(* CoDeSys 2.3.10.0 project: 20110511_Pantografo_2Ori_VNT15.pr6 *)
(* Libraries: STANDARD.LB6 5.6.98 11:03:02 *)

(* Global variable list: Global_Variables *)
VAR_GLOBAL CONSTANT
	MaxViti: BYTE:= 15;
	MaxFlange: BYTE:= 8;

	PiGreco: 			REAL := 3.14159265358979;					(*180 gradi*)
	PiGreco2: 		REAL:= 6.28318530717958;					(*360 gradi*)
	PiGrecoMezzi: 	REAL:= 1.5707963267949;					(*90 gradi*)
	PiGreco3Mezzi: 	REAL:= 4.71238898038469;					(*270 gradi*)
	Pigreco4i: 		REAL := 0.78539816339744830961566084581988;				(*45 gradi*)
	Pigreco3_8:		REAL:= 1.1780972450961724644234912687298;	(*60 gradi*)
	Rad2Gr:			REAL:= 57.295779513082320876798154814105; (*coeff. di conversione: 360 / (2*Pigreco)*)

	NonSvitabile:	BYTE:=	4;
	Riavvitare:	BYTE:=	3;
	Svitare:		BYTE:=	2;
	Good:		BYTE:=	1;
	NonEffettuata:	BYTE :=	0;

END_VAR
VAR_GLOBAL
	(*Comunicazione PFB*)
	Global_PFBComOK:	BOOL;
	Global_PFBComKO:	BOOL;

	(*Istanze Globali chiamate nel main*)
	Ist_MapA: 	MapA;
	Ist_MapE:	MapE;
	Ist_MapPFB:	MapPFB;


	(*Cicli*)
	Ist_CyclesMatching: 		CyclesMatching;
	Ist_CyclesDataReceiving:	CyclesDataReceiving;


	(*Macthing*)
	Screw: ARRAY [1..MaxViti] OF BOOL; (*array di esiti di metxhing dove l'indice è l'id_vite*)
	Prodotto:		Ricetta; (*ricetta punti vite*)
END_VAR

(* Data type in PAOLO *)
TYPE Avvitatura :
STRUCT
(*	NumMessaggio       : 	BYTE;
       	LunghezzaPacchetto : 	BYTE;
       	CodiceParametro    : 	BYTE;
       	free: 				BYTE;
	Shake:				Handshake;	(*WORD*)
*)
	ID_vite: 			BYTE;			(*identificativo della vite --> valutare il tipo: INT/STRING *)
 	Viti_Totali_Flangia : 	BYTE;
	ID_Flangia:		BYTE;			(*riferimento della flangia di appartenenza*)
	Chiave:			BYTE;			(*riferimento della chiave che va utilizzata su questa vite*)
	ProgAvvitatura: 	BYTE;			(*numero di programma da passare all'avvitatore per avvitate*)
	ProgRiavvitatura: 	BYTE;			(*numero di programma da passare all'avvitatore per riavvitare  *)
	ProgSvitatura:	BYTE;			(*numero di programma da passare all'avvitatore per svitare... se ZERO disabilita svitatura*)
	EsitoAvvitatura:	BYTE;			(*esito avvitatura 0 non effettuata 1 ok 2 scarto 3 svitato*)
(*esitoavvitatura sostituirebbe free2 della struttura scl*)
	Posizione:		Coordinate;
	TolleranzaR: 		REAL;			(*Raggio di tolleranza del punto*)
	TolleranzaZ: 		REAL;			(*Tolleranza Larga  in Altezza per entrare nello stato di Attesa Esito Avvitatura*)
	AltezzaMin:		REAL;			(*Tolleranza stretta Min Max*)
	AltezzaMax:		REAL;
(*       	riserva : ARRAY[76..123] OF BYTE;
*)
END_STRUCT
END_TYPE

(* Data type in PAOLO/ScambioDati/HEADER *)
TYPE Comandi :
STRUCT
	Matching:			BOOL;	(*comando di pantografo enable*)
	TxScrewingData:		BOOL;	(*comando di invio dati avvitatura*)
	RqstScrewingData:	BOOL;	(*comando di richiesta dati avvitatura*)
	ResettaEsitiAvvitature:	BOOL;
END_STRUCT
END_TYPE

(* Data type in PAOLO/ScambioDati/HEADER *)
TYPE CommunicationA :
STRUCT
	BeckMsgNum: 	BYTE;
	EchoPLCLifeBit:	BOOL;
	BeckLifeBit:		BOOL;
	Beck_ACK:		BOOL;
END_STRUCT
END_TYPE

(* Data type in PAOLO/ScambioDati/HEADER *)
TYPE CommunicationE :
STRUCT
	PlcMsgNum:	BYTE;
	PlcLifeBit:	BOOL;
	EchoBeckBit:	BOOL;	(*echo della mia uscita*)
	Plc_ACK:		BOOL;
END_STRUCT
END_TYPE

(* Data type in PAOLO *)
TYPE Coordinate :
STRUCT
	X:	REAL;		(*coordinate cartesiane x,y,z*)
	Y:	REAL;
	Z:	REAL;
	Angle:	REAL;	(*coordinate polari angolo,raggio*)
	Distance:REAL;
END_STRUCT
END_TYPE

(* Data type in Cicli *)
TYPE InputCiclo :
STRUCT
	Cm_ON:BOOL;
	HOLD:BOOL;
	STEP:BOOL;
END_STRUCT
END_TYPE

(* Data type *)
TYPE Lubbering :
STRUCT
	(*ID_Chiave:		BYTE;*)
	(*free:				BYTE;  su PLC *)
	AngoloMontaggio: REAL;	(*angolo di montaggio RISPETTO all'ANGOLO BRACCIO; 90 significa che con angolo polso a 0 e angolobraccio a 90, chiave parallela all'asse X*)
	Lub_Lunghezza:	REAL;	(*lungheza della chiave*)
END_STRUCT
END_TYPE

(* Data type in PAOLO/ScambioDati/HEADER *)
TYPE MacroStato :
STRUCT
	EsitiavvitatureResettati: BOOL;
	TxScrewingData: BOOL;
END_STRUCT
END_TYPE

(* Data type in PAOLO/ScambioDati/HEADER *)
TYPE MapHeaderA :
STRUCT
	Com:		CommunicationA;
	CmdECHO:	Comandi;
	Warn:		Warning;
	(*Alarms:*)
	MacroStati:	Macrostato;
END_STRUCT
END_TYPE

(* Data type in PAOLO/ScambioDati/HEADER *)
TYPE MapHeaderE :
STRUCT
(*allarmi*)
(*comunicazione*)
	Com:		CommunicationE;
	Cmd:		Comandi;
	WarnECHO:	Warning;(*opzionale lato PLC*)
END_STRUCT
END_TYPE

(* Data type in PAOLO/ScambioDati *)
TYPE MapPantoA :
STRUCT
	ParkingPosition:			BOOL;
	AbilitaAvvitatura:			BOOL;
	AbilitaSvitatura:			BOOL;
	AbilitaRiavvitatura:			BOOL;
	ViteNonSvitabile:			BOOL;
	Final_Position_OK:		BOOL;
	Final_Position_KO:		BOOL;
	AvvitatureTerminate:		BOOL;
	FrizioneComandata:		BOOL;
	Vite_in_Corso:			BYTE;
	ProgAvvitatura:			BYTE;
	Chiave:					BYTE; (*Codice chiave da usare per la vite*)
	VitiEffettuate:				BYTE;
	X:						REAL;
	Y:						REAL;
	Z:						REAL;
END_STRUCT
END_TYPE

(* Data type in PAOLO/ScambioDati *)
TYPE MapPantoE :
STRUCT
	StartPls:				BOOL;
	Avvitatore_EsitoOK:	BOOL;
	Avvitatore_EsitoKO:	BOOL;
	Avvitatura_InCorso:	BOOL;
	Avvitatura_Fine:		BOOL;
	Avvitatura_Ripeti:		BOOL;
	ECHO_Viti_Effettuate:	BYTE;
	Viti_Totali_Flangia:	BYTE;
	FlangiaInCorso:		BYTE;
	AngoloPallet:			REAL;	(*link se è abilitato il piano rotante*)
	ProgAvvitGenerico:	BYTE;	(*usato se disabilitati check z zfinale e piano *)
END_STRUCT
END_TYPE

(* Data type in PAOLO/ScambioDati *)
TYPE MapPantoParE :
STRUCT
(*globali*)
	Globali:	ParametriGlobali;
(*machine*)
	Macchina:	ParametriMacchina;
(*sensori*)
	Sensori:		ParametriSensori;
END_STRUCT
END_TYPE

(* Data type in PAOLO/ScambioDati *)
TYPE MapScrewingE :
STRUCT
	FlangiaInviata:		BYTE;
	Viti_Totali_Flangia:	BYTE;
	Id_ViteInviata:			BYTE;
	ID_Chiave:			BYTE;
	ProgAvvitatura:		BYTE;
	ProgRiavvitatura:		BYTE;
	ProgSvitatura:		BYTE;
	X:					REAL;
	Y:					REAL;
	Z:					REAL;
	TollR:				REAL;
	TollZ:				REAL;
	ZMin:				REAL;
	ZMax:				REAL;
END_STRUCT
END_TYPE

(* Data type in Cicli *)
TYPE OutputCiclo :
STRUCT
	CicloInCorso:BOOL;
	CicloTerminatoOK:BOOL;
	CicloTerminatoKO:BOOL;
	Stato:INT;
	Messaggio:INT;
END_STRUCT
END_TYPE

(* Data type in PAOLO/ScambioDati/Ricetta_ *)
TYPE ParametriGlobali :
STRUCT
	ProgrammaSvitatura: 	BYTE;
	SvitaturaSuScarto:		BOOL;
	CheckZ:				BOOL;
	CheckZfinale:			BOOL;
	PianoRotanteAttivo:	BOOL;
	Lub1_enable:			BOOL;	(*abilitazione chiave 1*)
	Lub2_enable:			BOOL;	(*abilitazione chiave 2*)
	CheckPianoXY:		BOOL;
	ScrewSequenceActive:	BOOL;
END_STRUCT
END_TYPE

(* Data type in PAOLO/ScambioDati/Ricetta_ *)
TYPE ParametriMacchina :
STRUCT
	AsseVerticaleX:	REAL;
	AsseVerticaleY:	REAL;
	L1_lunghezza:	REAL;
	L1_Angolo:		REAL;
	OscillAvvitatore:	REAL;
	Lub:				ARRAY [1..2] OF Lubbering;
	(*Lub1:			Lubbering;
	Lub2:			Lubbering;*)
	ParkZone:		Parcheggio;
END_STRUCT
END_TYPE

(* Data type in PAOLO/ScambioDati/Ricetta_ *)
TYPE ParametriSensori :
STRUCT
	AngoloBraccio:	Sensore;
	Z:				Sensore;
	EstBraccio:		Sensore;
	Z2:				Sensore;
	Polso:			Sensore;
END_STRUCT
END_TYPE

(* Data type *)
TYPE Parcheggio :
STRUCT
	AllungMax:	REAL;
	Allungmin:	REAL;
	AngoloMax:	REAL;
	AngoloMin:   	REAL;
	AltezzaMin: 	REAL;
END_STRUCT
END_TYPE

(* Data type in PAOLO *)
TYPE PolarCoord :
STRUCT
	Angle:	REAL;	(*coordinate polari*)
	Distance:REAL;
END_STRUCT
END_TYPE

(* Data type in PAOLO/ScambioDati/Ricetta_ *)
TYPE Ricetta :
STRUCT
	PuntoVite: ARRAY [1..MaxFlange, 1..MaxViti] OF	Avvitatura;	(*partiamo dall'indice vite ZERO anche se non viene usato per evitare errori di locazione array*)
(*	Viti_totali :			BYTE;
	Viti_Effettuate:			BYTE;*)
END_STRUCT
END_TYPE

(* Data type *)
TYPE Sensore :
STRUCT
	Gain:	REAL;
	Offset:	REAL;
END_STRUCT
END_TYPE

(* Data type in PAOLO/ScambioDati/HEADER *)
TYPE Warning :
STRUCT
	RicettaVuota:				BOOL;
	OffsetMancante: 			BOOL;
	ParametriLubMancanti: 	BOOL;
	FuoriIngombroInconsistente:BOOL;
	AngleArmsGainMissing: 	BOOL;
	ZAxisGainMissing:			BOOL;
	LengthArmsGainMissing: 	BOOL;
	NoGainAsseZ2:			BOOL;
	NoGainPolso:			BOOL;
END_STRUCT
END_TYPE

(* POU MAIN, ST *)
PROGRAM MAIN
VAR
	sys: 	Systems;

END_VAR
(*istanze Mapping*)
Ist_MapE();

Ist_MapPFB();

(*istanza cicli*)
Cycles();

(*istanza sitema*)
sys();

Ist_MapA();

(*%QX0.0:=TRUE;
%QX0.1:=TRUE;
%QX0.2:=TRUE;
%QX0.3:=TRUE;*)
END_PROGRAM

(* POU Systems, ST *)
FUNCTION_BLOCK Systems(*struttura System:
								LIFE BIT CHECK
								PANTOGRAFO
								PARKING ZONE
								MATCHING
								 test PANTOGRAFO
								GESTIONE WARNING*)
VAR_INPUT
END_VAR
VAR_OUTPUT
END_VAR
VAR
	(*PFB_Communication : FB_SystemLifeBitCheck;*)
	LifeBitSystem: LifeBit;
	PlcLifeBitOLD: BOOL;
	TimeOUT: TON;
	Fase:	INT;	(*idea alternativa a Pagina*)
	Pantografo:	FB_SystemPantoNEW;(*FB_SystemPanto;*)

	PrimaViteDaCercare : BYTE;

	(*matching*)
	(*utilizzato variabile Screw array of bool di esiti di matching dove l'indice è l'id_vite*)
	iVite:	BYTE;
	iFlangia:	BYTE;
	Utensile: BYTE;
	MemFlangia: BYTE;
	(*EsitiResettati: BOOL;*)
	UltimaFlangia: BYTE;
	ActualPosition:	Coordinate;(*Coord;*)		(*posizione attuale no lub coord X ,Y e Z*)
	ViteTrovata:		BYTE;
	UltimaViteRegistrata:	BYTE;
	ViteAvvitabile:	BOOL;
	ViteIncrementata:	BOOL;
	Ist_Match:		FB_Std_Match;
	DisabledMatchingState: BOOL;
	Vite_in_CorsoOLD: BYTE; (*vite del clock precedente*)
	(*PARKING ZONE*)
	ParkingZone:		Coordinate;
(*	ParkingMatch:	FB_Std_Match;	(*istanza per la verifica della zona di parcheggio*)*)

	(*accodamento avvitatura*)


(*TEST*)
	TestMatch: BOOL;
	TestMatch_CheckZ: BOOL;
	TestMatch_CheckZfinale: BOOL;
	TestMatch_CheckPianoXY: BOOL;
(*	a: BYTE;
	b:BYTE;
*)

	TestPanto: BOOL;
			L1_Lungh:REAL;
			L1_Angle:REAL;
			Est_Braccio:REAL;
			Rad_Braccio:REAL;
			L1Angle:REAL;
			ScrewerXRif:REAL;
			ScrewerYRif:REAL;
			ZBraccio:REAL;
			ZBraccio2:REAL;
			Lub1_en:BOOL;
			Lub2_en:BOOL;
			PianoRot_en:BOOL;
			RadPiano:REAL;
			Rad_Polso:REAL;
			Chiave1:Lubbering;
			Chiave2:Lubbering;
			OrigineX:REAL;
			OrigineY:REAL;
			OrigineZ:REAL;
	(***)
END_VAR
(*costanti messe in Globali
	Scarto:		BYTE:= 2;
	Good: 		BYTE:= 1;
	NonEffettuata :BYTE := 0;*)
(*---------------------------LIFE BIT CHECK-------------------------*)
	(*--------Istanza FB_SystemCommunication------*)
(*comunico al partner che sono vivo*)
LifeBitSystem(NumCicli:= 5, LifeBit=> Ist_MapPFB.HeaderA.Com.BeckLifeBit);

(*verifico che il partner non sia morto e inizio a contare quando non cambia di stato il plclifebit*)
TimeOUT(IN:= Ist_MapPFB.HeaderE.Com.PlcLifeBit =  PlcLifeBitOLD,
		PT:= t#7s);
PlcLifeBitOLD:= Ist_MapPFB.HeaderE.Com.PlcLifeBit;
Global_PFBComOK:= NOT TimeOUT.Q;
Global_PFBComKO:= TimeOUT.Q;

Ist_MapPFB.HeaderA.Com.EchoPLCLifeBit:= Ist_MapPFB.HeaderE.Com.PlcLifeBit;


(*Gestione Fase a mò di pagina per ora bypassata*)
IF Global_PFBComOK OR Global_PFBComKO
THEN
	Fase:= 1;
END_IF
(*
IF Global_PFBComKO
THEN
	Fase:= 0;
END_IF
*)

IF TestPanto
THEN
	Fase:= 253;
END_IF
(*-------------------fine ------LIFE BIT CHECK-------------------------*)

CASE Fase OF
0: 	(*GESTIONE Comunicazione Caduta-> resettare uscite??? VALUTARE*)
(*inizio case Fase=0*)
;
(*fine case Fase=0*)

1:	(*Global_PFBComOK -> trasportare qui ciò che prima era in system*)
(*inizio case Fase=1*)

(*------------------------------------------------- PANTOGRAFO-----------------*)

(****NEW FB_System Pantografo****)

Pantografo(
	L1_Lungh:=  		Ist_MapPFB.PantoParE.Macchina.L1_lunghezza,
	L1_AngleType:= 	Ist_MapPFB.PantoParE.Macchina.L1_Angolo ,
	Braccio_Est:=		Ist_MapE.EstBraccio,
	Braccio_Rad:= 	Ist_MapE.RadBraccio,
	ZBraccio:= 		Ist_MapE.Z,
	ZBraccio2:= 		Ist_MapE.Z_Braccio2,
	RadPiano:= 		SEL(Ist_MapPFB.PantoParE.Globali.PianoRotanteAttivo, 0, Ist_MapPFB.PantoE.AngoloPallet /Rad2Gr),
	Polso_Rad:= 		Ist_MapE.RadPolso,
	Chiave1:= 		Ist_MapPFB.PantoParE.Macchina.Lub[1],
	Chiave2:= 		Ist_MapPFB.PantoParE.Macchina.Lub[2],
	Lub1_en:= 		Ist_MapPFB.PantoParE.Globali.Lub1_enable,
	Lub2_en:= 		Ist_MapPFB.PantoParE.Globali.Lub2_enable,
	PianoRot_en:= 	Ist_MapPFB.PantoParE.Globali.PianoRotanteAttivo,
	X_Offset:= 		Ist_MapPFB.PantoParE.Macchina.AsseVerticaleX,
	Y_Offset:= 		Ist_MapPFB.PantoParE.Macchina.AsseVerticaleY);

(*assegno i valori  XYZ  alle Uscite*)
Ist_MapPFB.PantoA.X:= Pantografo.ActualPosition.X;
Ist_MapPFB.PantoA.Y:= Pantografo.ActualPosition.Y;
Ist_MapPFB.PantoA.Z:= Pantografo.ActualPosition.Z;
(*-------------------------------------------------------------FINE PANTOGRAFO-----------------*)

(*------------------------------------------------------PARKING ZONE------------------------------------------*)

Ist_MapPFB.PantoA.ParkingPosition:= 	(Ist_MapE.RadBraccio > (Ist_MapPFB.PantoParE.Macchina.ParkZone.AngoloMin / Rad2Gr)) AND
								  	(Ist_MapE.RadBraccio < (Ist_MapPFB.PantoParE.Macchina.ParkZone.AngoloMax / Rad2Gr)) AND
							           	(Ist_MapE.EstBraccio < Ist_MapPFB.PantoParE.Macchina.ParkZone.AllungMax) AND
								  	(Ist_MapE.EstBraccio > Ist_MapPFB.PantoParE.Macchina.ParkZone.AllungMin) AND
								 	(Pantografo.ActualPosition.Z > Ist_MapPFB.PantoParE.Macchina.ParkZone.AltezzaMin) ;

(*valutare se usare l'area stretta - sottoinsieme dell'area larga perchè valuta anche Zmin e Zmax*)
(*--FINE------------------------------------------------PARKING ZONE------------------------------------------*)


(*-------------------------------------------------------------------- MATCHING-----------------*)
(*----------------Comando di resetta Esiti----------------- VALUTARE un handshake verso il partner per lo stato *)
IF Ist_MapPFB.HeaderE.Cmd.ResettaEsitiAvvitature
(*AND NOT Ist_MapPFB.HeaderA.MacroStati.EsitiavvitatureResettati*)
THEN
	FOR iFlangia:=1 TO MaxFlange
	DO
		FOR iVite:= 1 TO MaxViti
		DO
			Prodotto.PuntoVite[iFlangia,iVite].EsitoAvvitatura:= NonEffettuata;
			UltimaViteRegistrata :=NonEffettuata;
		END_FOR(*viti*)
	END_FOR(*flange*)
	Ist_MapPFB.PantoA.VitiEffettuate:= NonEffettuata;
END_IF
Ist_MapPFB.HeaderA.MacroStati.EsitiavvitatureResettati :=Ist_MapPFB.HeaderE.Cmd.ResettaEsitiAvvitature;	(*appoggio per il rilevamento del fronte positivo*)

(*se sono in test assegno Test_iFlangia altrimenti il mapping da PFB*)
iFlangia:= Ist_MapPFB.PantoE.FlangiaInCorso;
IF iFlangia <= 0
THEN
	iFlangia:= 1;
END_IF

IF iFlangia <> MemFlangia THEN (* init Utensile al cambio della flangia *)
	Utensile := Prodotto.PuntoVite[iFlangia, 1].Chiave;
END_IF;

IF UltimaFlangia <> iFlangia	(*resetto le viti effettuate se si cambia flangia ma ATTENZIONE così salto vititerminate*)
(*AND NOT UnPasso*)
THEN
	Ist_MapPFB.PantoA.VitiEffettuate:=0;
END_IF
IF Ist_MapPFB.PantoE.Viti_Totali_Flangia > Ist_MapPFB.PantoA.VitiEffettuate(*OLD Prodotto.Viti_totali > Prodotto.Viti_Effettuate*)
(*AND NOT UnPasso*)
THEN
	Ist_MapPFB.PantoA.AvvitatureTerminate:= FALSE; (*Reset*)
	UltimaFlangia:= iFlangia;	(*segno l'ultima flangia in corso*)

	IF ViteTrovata = 0 THEN
		ViteTrovata := 1; (* se non già trovata una vite provo con la prima *)
		PrimaViteDaCercare := 2;
	ELSE
		PrimaViteDaCercare := 1;
	END_IF
	iVite := ViteTrovata;
	Ist_Match (	Actualpoint:= 		Pantografo.ActualPosition,							(*posizione attuale di tipo coordinate XYZ+Angolo+R*)
				Point2Match:= 	Prodotto.PuntoVite[iFlangia, iVite].Posizione,			(*coordinate del punto da "matchare"*)
				R_Toll:=			Prodotto.PuntoVite[iFlangia, iVite].TolleranzaR,			(*raggio di tolleranza del punto "matchare"*)
				Z_Toll:=			Prodotto.PuntoVite[iFlangia, iVite].TolleranzaZ,			(*tolleranza di Z del punto "matchare" -> tolleranza simmetrica per lo start avvitatura*)
				Z_Min:=			Prodotto.PuntoVite[iFlangia, iVite].AltezzaMin,			(*altezza minima per il check della posizione a fine avvitatura *)
				Z_Max:=  		Prodotto.PuntoVite[iFlangia, iVite].AltezzaMax,			(*altezza massima per il check della posizione a fine avvitatura *)
				ZCheck:=		SEL(TestMatch, Ist_MapPFB.PantoParE.Globali.CheckZ, TestMatch_CheckZ),	(*abilitazione controllo altezza per lo start avvitatura*)
				ZCheckFinale:=  	SEL(TestMatch, Ist_MapPFB.PantoParE.Globali.CheckZfinale, TestMatch_CheckZfinale),(*abilitazione controllo della posizione a fine avvitatura*)
				PianoCheck:= 	SEL(TestMatch, Ist_MapPFB.PantoParE.Globali.CheckPianoXY, TestMatch_CheckPianoXY),(*abilitazione controllo XY per lo start avvitatura*)
				oscill:=			Ist_MapPFB.PantoParE.Macchina.OscillAvvitatore,		(*parametro di ulteriore tolleranza di oscillazione*)
				oscill_Default:=	0,												(*valore di deflault della tolleranza di oscillazione*)
				oscill_Ev:= 		Ist_MapPFB.PantoE.Avvitatura_InCorso,
				EsitoAvvitatura:=	Prodotto.PuntoVite[iFlangia, iVite].EsitoAvvitatura);				(*evento per lo switching del valore di tolleranza oscillazione*)

	(*valutazione area larga*)
	IF Ist_Match.AreaLarga_OK			(*se trovo una vite nell'area larga  mi segno l'id_vite e forzol'index ad viti_totali + 1*)
	THEN
		IF NOT Ist_Match.PianoCheck
		THEN
			ViteTrovata:= Ist_MapPFB.PantoA.VitiEffettuate + 1;
		ELSE
			ViteTrovata:= iVite;
		END_IF
	ELSE
		(*-----------------------inizio scansione viti-------------------*)
		iVite:= PrimaViteDaCercare;
		REPEAT
		(*FOR iVite:= 1 TO Ist_MapPFB.PantoE.Viti_Totali_Flangia	se trovo una vite nell'area larga  mi segno l'id_vite e forzol'index ad viti_totali + 1*)
		(*DO													altrimenti ViteTrovata resta al valore di init*)
			(*init flag*)
			ViteTrovata:= 0;
			(*Istanza di Matching con la posizione attuale*)
			Ist_Match (	Actualpoint:= 		Pantografo.ActualPosition,							(*posizione attuale di tipo coordinate XYZ+Angolo+R*)
						Point2Match:= 	Prodotto.PuntoVite[iFlangia, iVite].Posizione,			(*coordinate del punto da "matchare"*)
						R_Toll:=			Prodotto.PuntoVite[iFlangia, iVite].TolleranzaR,			(*raggio di tolleranza del punto "matchare"*)
						Z_Toll:=			Prodotto.PuntoVite[iFlangia, iVite].TolleranzaZ,			(*tolleranza di Z del punto "matchare" -> tolleranza simmetrica per lo start avvitatura*)
						Z_Min:=			Prodotto.PuntoVite[iFlangia, iVite].AltezzaMin,			(*altezza minima per il check della posizione a fine avvitatura *)
						Z_Max:=  		Prodotto.PuntoVite[iFlangia, iVite].AltezzaMax,			(*altezza massima per il check della posizione a fine avvitatura *)
						ZCheck:=		SEL(TestMatch, Ist_MapPFB.PantoParE.Globali.CheckZ, TestMatch_CheckZ),	(*abilitazione controllo altezza per lo start avvitatura*)
						ZCheckFinale:=  	SEL(TestMatch, Ist_MapPFB.PantoParE.Globali.CheckZfinale, TestMatch_CheckZfinale),(*abilitazione controllo della posizione a fine avvitatura*)
						PianoCheck:= 	SEL(TestMatch, Ist_MapPFB.PantoParE.Globali.CheckPianoXY, TestMatch_CheckPianoXY),(*abilitazione controllo XY per lo start avvitatura*)
						oscill:=			Ist_MapPFB.PantoParE.Macchina.OscillAvvitatore,		(*parametro di ulteriore tolleranza di oscillazione*)
						oscill_Default:=	0,												(*valore di deflault della tolleranza di oscillazione*)
						oscill_Ev:= 		Ist_MapPFB.PantoE.Avvitatura_InCorso,
						EsitoAvvitatura:=	Prodotto.PuntoVite[iFlangia, iVite].EsitoAvvitatura);		(*evento per lo switching del valore di tolleranza oscillazione*)

			(*valutazione area larga*)
			IF Ist_Match.AreaLarga_OK			(*se trovo una vite nell'area larga  mi segno l'id_vite e forzol'index ad viti_totali + 1*)
			THEN
				IF NOT Ist_Match.PianoCheck
				THEN
					ViteTrovata:= Ist_MapPFB.PantoA.VitiEffettuate + 1;
				ELSE
					ViteTrovata:= iVite;
				END_IF
				iVite:= Ist_MapPFB.PantoE.Viti_Totali_Flangia;		(*FORZO l'uscita dal ciclo FOR*)
			END_IF
			iVite := iVite + 1;
		UNTIL iVite > Ist_MapPFB.PantoE.Viti_Totali_Flangia
		END_REPEAT
		(*-----------------------fine    scansione viti-------------------*)
	END_IF

	Screw:= FC_InitArea(Screw);	(*init array "ombra" di bool *)
	ViteAvvitabile:= FALSE;(*init/reset ViteAvvitabile*)
	IF ViteTrovata<> 0	(*Trovata vite iesima in AreaLarga - in caso di Match con controlli disabilitati ViteTrovata sarà sempre 1 cioè la prima istanza con AreaLarga_OK*)
	THEN
		ViteAvvitabile :=FC_Avvitabile(id_avv:=ViteTrovata , id_flangia:= iFlangia);(*SET*)
		IF Ist_Match.AreaLarga_OK AND ViteAvvitabile
		THEN
			(*genero l'evento che crea  lo start ciclo di matching (e lo mantiene in ciclo)-> segno la vite trovata *)
			Screw[ViteTrovata]:= TRUE;
		END_IF
	END_IF(*fin ViteTrovata<>0*)

	(*----VALUTAZIONE RISULTATI in base agli stati del Ciclo Matching------------------*)

	(*--------------Stato <0> : StartAvvitatura---------*)
	IF Ist_CyclesMatching.Stato = 0 		(*ABILITA AVVITATURA: Stato di Viti Avvitabili e  Start Avvitatura quindi -> già valutati posizione e avvitabilità*)
	THEN
		Ist_MapPFB.PantoA.ProgAvvitatura := 	0;
		Ist_MapPFB.PantoA.Vite_in_Corso :=		0; (*oppure -> Prodotto.PuntoVite[iFlangia,ViteTrovata].ID_vite*)
		Ist_MapPFB.PantoA.AbilitaAvvitatura :=	FALSE;
		Ist_MapPFB.PantoA.AbilitaSvitatura := 	FALSE;
		Ist_MapPFB.PantoA.AbilitaRiavvitatura := 	FALSE;
		Ist_MapPFB.PantoA.ViteNonSvitabile := 	FALSE;
	END_IF (*fine stato 0*)

	(*--------------Stato <10> : StartAvvitatura---------*)
	IF Ist_CyclesMatching.Stato = 10 		(*ABILITA AVVITATURA: Stato di Viti Avvitabili e  Start Avvitatura quindi -> già valutati posizione e avvitabilità*)
	THEN
		IF ViteTrovata <> 0 THEN
			Ist_MapPFB.PantoA.Vite_in_Corso	:=	ViteTrovata; (*oppure -> Prodotto.PuntoVite[iFlangia,ViteTrovata].ID_vite*)
			Utensile							:= 	Prodotto.PuntoVite[iFlangia,ViteTrovata].Chiave;
			(*controllo se la vite era stata scartata al ciclo precedente*)
			IF Prodotto.PuntoVite[iFlangia,ViteTrovata].EsitoAvvitatura = Svitare
			THEN
				Ist_MapPFB.PantoA.AbilitaAvvitatura:=	TRUE;
				Ist_MapPFB.PantoA.AbilitaSvitatura:= 	TRUE;
				Ist_MapPFB.PantoA.AbilitaRiavvitatura := 	FALSE;
				Ist_MapPFB.PantoA.ViteNonSvitabile := 	FALSE;
				(*restituisco il programma di svitatura*)
				Ist_MapPFB.PantoA.ProgAvvitatura:= Prodotto.PuntoVite[iFlangia,ViteTrovata].ProgSvitatura;
			ELSIF Prodotto.PuntoVite[iFlangia,ViteTrovata].EsitoAvvitatura = Riavvitare
			THEN
				(*consegna al PLC di: Vite "Matchata", relativo ProgAvvitatura, setto TRUE a Abilita Avvitatura; NOTA: se sono nello stato di Matching disabilitato consegno il prog generico*)
				Ist_MapPFB.PantoA.AbilitaAvvitatura:=	TRUE;
				Ist_MapPFB.PantoA.AbilitaSvitatura:= 	FALSE;
				Ist_MapPFB.PantoA.AbilitaRiavvitatura :=	TRUE;
				Ist_MapPFB.PantoA.ViteNonSvitabile := 	FALSE;
				Ist_MapPFB.PantoA.ProgAvvitatura:= Prodotto.PuntoVite[iFlangia,ViteTrovata].ProgRiavvitatura;
			ELSIF Prodotto.PuntoVite[iFlangia,ViteTrovata].EsitoAvvitatura = NonEffettuata  (* CARICA PROGRAMMA AVVITATURA AVVITA VITE  *)
			THEN
				(*consegna al PLC di: Vite "Matchata", relativo ProgAvvitatura, setto TRUE a Abilita Avvitatura; NOTA: se sono nello stato di Matching disabilitato consegno il prog generico*)
				Ist_MapPFB.PantoA.AbilitaAvvitatura:=	TRUE;
				Ist_MapPFB.PantoA.AbilitaSvitatura:= 	FALSE;
				Ist_MapPFB.PantoA.AbilitaRiavvitatura := 	FALSE;
				Ist_MapPFB.PantoA.ViteNonSvitabile :=	FALSE;
				Ist_MapPFB.PantoA.ProgAvvitatura:= Prodotto.PuntoVite[iFlangia,ViteTrovata].ProgAvvitatura;
			ELSE
				Ist_MapPFB.PantoA.AbilitaAvvitatura:= 	Ist_MapPFB.PantoE.Avvitatura_Ripeti;
				Ist_MapPFB.PantoA.AbilitaSvitatura:= 	FALSE;
				Ist_MapPFB.PantoA.AbilitaRiavvitatura := 	FALSE;
				Ist_MapPFB.PantoA.ViteNonSvitabile := 	NOT Ist_MapPFB.PantoE.Avvitatura_Ripeti;
				Ist_MapPFB.PantoA.ProgAvvitatura:= Prodotto.PuntoVite[iFlangia,ViteTrovata].ProgAvvitatura;
			END_IF
		END_IF
	END_IF (*fine stato 10*)
(*????valutazione ed evoluzione nello stato 15*)

	(*--------------Stato <15> : StartAvvitatura---------*)
	IF Ist_CyclesMatching.Stato = 15 		(*ABILITA AVVITATURA: Stato di Viti Avvitabili e  Start Avvitatura quindi -> già valutati posizione e avvitabilità*)
	THEN
		IF NOT Ist_Match.AreaLarga_OK							(*se non sono sull'area di avvitatura*)
		OR Ist_MapPFB.PantoA.Vite_in_Corso <> Vite_in_CorsoOLD 	(*o senon sono  sulla vite del clock precedente*)
		THEN
			Ist_MapPFB.PantoA.AbilitaAvvitatura	:=	FALSE; (*RESET*)
			Ist_MapPFB.PantoA.AbilitaSvitatura	:=	FALSE;
			Ist_MapPFB.PantoA.AbilitaRiavvitatura := 	FALSE;
			Ist_MapPFB.PantoA.ViteNonSvitabile := 	FALSE;
			Ist_MapPFB.PantoA.ProgAvvitatura := 	0;
		END_IF
	END_IF (*fine stato 15*)

	(*-------------Stato <30> Esito FineAvvitatura OK -> CheckFinalPosition*)
	IF Ist_CyclesMatching.Stato = 30
	THEN
		IF  Ist_Match.AreaStretta_OK
		THEN
			Ist_MapPFB.PantoA.Final_Position_OK:= TRUE; (*SET*)

			IF NOT ViteIncrementata  AND (UltimaViteRegistrata <>  ViteTrovata) AND (NOT Ist_MapE.StartPls OR NOT Ist_MapPFB.PantoParE.Globali.ScrewSequenceActive)
				(*soluzione per operare un solo incremento*)
			THEN
				Ist_MapPFB.PantoA.VitiEffettuate:=  Ist_MapPFB.PantoA.VitiEffettuate + 1;
				ViteIncrementata:= TRUE;
				Prodotto.PuntoVite[iFlangia,ViteTrovata].EsitoAvvitatura := Good;
				UltimaViteRegistrata:= ViteTrovata;
			END_IF
		ELSE
			Ist_MapPFB.PantoA.Final_Position_KO:= TRUE; (*SET*)
		END_IF
	ELSE
		ViteIncrementata:= FALSE; (*reset*)
	END_IF(*fine stato 30*)

	(*---------------Stato <37> :  Attesa RESET da parte del PLC -------------*)
	IF Ist_CyclesMatching.Stato = 60
	THEN
		(*RESET abilitazioni*)
		(*Ist_MapPFB.PantoA..AbilitaAvvitatura := FALSE;*)
		Ist_MapPFB.PantoA.Final_Position_OK:= 	FALSE;
		Ist_MapPFB.PantoA.ProgAvvitatura:= 	NonEffettuata;
		Ist_MapPFB.PantoA.AbilitaAvvitatura	:=	FALSE; (*RESET*)
		Ist_MapPFB.PantoA.AbilitaSvitatura	:=	FALSE;
		Ist_MapPFB.PantoA.AbilitaRiavvitatura := 	FALSE;
		Ist_MapPFB.PantoA.ViteNonSvitabile := 	FALSE;
	END_IF (*fine stato60*)

	IF Ist_CyclesMatching.Stato = 45 (*OR Ist_CyclesMatching.Stato = 59*)
	THEN
		(*AbilitaAvvitatura -> Resta invariato*)
		Ist_MapPFB.PantoA.Final_Position_KO:= FALSE; (*SET*)
		IF  Prodotto.PuntoVite[iFlangia,ViteTrovata].ProgSvitatura <> 0
		THEN
			Prodotto.PuntoVite[iFlangia,ViteTrovata].EsitoAvvitatura := Svitare;
			Ist_MapPFB.PantoA.AbilitaAvvitatura:=	TRUE;
			Ist_MapPFB.PantoA.AbilitaSvitatura:= 	TRUE;
			Ist_MapPFB.PantoA.AbilitaRiavvitatura := 	FALSE;
			Ist_MapPFB.PantoA.ViteNonSvitabile := 	FALSE;
			(*Vite_in_Corso resta invariata*)
			(*il prog di avvitatura si trasfoema nel programma di svitatura*)
			Ist_MapPFB.PantoA.ProgAvvitatura:= Prodotto.PuntoVite[iFlangia,ViteTrovata].ProgSvitatura ;
		ELSE
			Prodotto.PuntoVite[iFlangia,ViteTrovata].EsitoAvvitatura := NonSvitabile;
			Ist_MapPFB.PantoA.AbilitaAvvitatura	:=	FALSE; (*RESET*)
			Ist_MapPFB.PantoA.AbilitaSvitatura	:=	FALSE;
			Ist_MapPFB.PantoA.AbilitaRiavvitatura := 	FALSE;
			Ist_MapPFB.PantoA.ViteNonSvitabile := 	TRUE;
			Ist_MapPFB.PantoA.ProgAvvitatura:= 0;
		END_IF

		IF NOT Ist_Match.AreaLarga_OK							(*se non sono sull'area di avvitatura*)
		OR Ist_MapPFB.PantoA.Vite_in_Corso <> Vite_in_CorsoOLD 	(*o senon sono  sulla vite del clock precedente*)
		THEN
			Ist_MapPFB.PantoA.AbilitaAvvitatura	:=	FALSE; (*RESET*)
			Ist_MapPFB.PantoA.AbilitaSvitatura	:=	FALSE;
			Ist_MapPFB.PantoA.AbilitaRiavvitatura := 	FALSE;
			Ist_MapPFB.PantoA.ViteNonSvitabile := 	FALSE;
		END_IF
	END_IF(*fine stato45*)

	(* Filippone 17/12/2010 *)
	IF Ist_CyclesMatching.Stato = 50
	THEN
		IF  Prodotto.PuntoVite[iFlangia,ViteTrovata].ProgSvitatura <> 0
		THEN
			Prodotto.PuntoVite[iFlangia,ViteTrovata].EsitoAvvitatura := Riavvitare;
		END_IF;
	END_IF(*fine stato50*)


	(*Stato <55> :  Svitatura Terminata -> RST dei SET dello Stato 45*)
	IF Ist_CyclesMatching.Stato = 55
	THEN
		Ist_MapPFB.PantoA.AbilitaAvvitatura	:=	FALSE; (*RESET*)
		Ist_MapPFB.PantoA.AbilitaSvitatura	:=	FALSE;
		Ist_MapPFB.PantoA.AbilitaRiavvitatura := 	FALSE;
		Ist_MapPFB.PantoA.ViteNonSvitabile := 	FALSE;
		Ist_MapPFB.PantoA.ProgAvvitatura:= 	NonEffettuata;
		Ist_MapPFB.PantoA.Vite_in_Corso:= 		NonEffettuata;
		Ist_MapPFB.PantoA.Final_Position_KO:= 	FALSE;
	END_IF(*fine stato45*)

(*Gestione del Fine Ciclo*)
	IF NOT Ist_CyclesMatching.CicloInCorso	(*Fase di  Reset cmd  MODIFICARE il Reset di abilita avvityatura qui*)
	THEN
		Ist_MapPFB.PantoA.ProgAvvitatura := 	NonEffettuata;		(*RST anche  in ramo Buono-> Stato37  ramo Scarto-> Stato45 *)
		Ist_MapPFB.PantoA.Vite_in_Corso:= 		NonEffettuata;		(*VALUTARE se mi serve*)
		Ist_MapPFB.PantoA.Final_Position_OK := 	FALSE;			(*RESETTATO in ramo Buono-> Stato37  *)
		Ist_MapPFB.PantoA.Final_Position_KO := 	FALSE;			(*RESETTATO in Stato*)
		Ist_MapPFB.PantoA.AbilitaAvvitatura :=	FALSE;
		Ist_MapPFB.PantoA.AbilitaSvitatura := 	FALSE;
		Ist_MapPFB.PantoA.AbilitaRiavvitatura := 	FALSE;
		Ist_MapPFB.PantoA.ViteNonSvitabile := 	FALSE;
	END_IF
ELSE(*fine viti da avvitare*)
	Utensile:=				 				0;
	Ist_MapPFB.PantoA.AvvitatureTerminate:=	TRUE;	(*SET*)
	Ist_MapPFB.PantoA.AbilitaAvvitatura:= 		FALSE;	(*RESET  - OTTIMIZZARE CODICE idea bistabili*)
	Ist_MapPFB.PantoA.AbilitaSvitatura := 		FALSE;
	Ist_MapPFB.PantoA.AbilitaRiavvitatura := 		FALSE;
	Ist_MapPFB.PantoA.ViteNonSvitabile := 		FALSE;
END_IF(*Viti Terminate*)

Ist_MapPFB.PantoA.Chiave := Utensile;
MemFlangia := iFlangia;

Vite_in_CorsoOLD:= Ist_MapPFB.PantoA.Vite_in_Corso;


(*-------------------------------------------------------------FINE MATCHING-----------------*)

(*-----------------------------------GESTIONE ACCODAMENTO AVVITATURE-----------------------------*)
Ist_MapPFB.HeaderA.MacroStati.TxScrewingData:= Ist_MapPFB.HeaderE.Cmd.TxScrewingData;
IF Ist_CyclesDataReceiving.Stato = 20 (*Stati <20> : Fase di Accodamento e inizio Handshake2*)
THEN
	Ist_MapPFb.EsitoAccodamento:= FC_PuntoViteAppend(); (*Set Esito*)
	ViteTrovata := 0;
END_IF
IF NOT Ist_CyclesDataReceiving.CicloInCorso(*Stati <60> : Fine Ciclo OR Not in Cycle*)
THEN
	Ist_MapPFB.EsitoAccodamento:= 0; (*Reset Esito*)
	(*Ist_MapPFB.HeaderA.Com.BeckMsgNum:= 0; (*gestito anchde nel  ciclo*)	(*Reset Msg Num per ogni invio singola vite per evitare il 255 - 0  0 = 255 + 1?? in byte si ma in in no  *)
*)
END_IF

(*------fine-------------------------GESTIONE ACCODAMENTO AVVITATURE-----------------------------*)

(*fine case Fase=1*)

253: ;(*test pantografo*)
(*------------------------------------------------- test PANTOGRAFO-----------------*)

(*-------------------------------------------------------------FINE PANTOGRAFO-----------------*)
END_CASE

(*---------------------------GESTIONE WARNING-----------------*)

Ist_MapPFB.HeaderA.Warn.RicettaVuota:=		Prodotto.PuntoVite[1,1].ProgAvvitatura = 0; 	(*RicettaInconsistente*)


Ist_MapPFB.HeaderA.Warn.OffsetMancante:=		Ist_MapPFB.PantoParE.Macchina.AsseVerticaleX = 0
										OR	Ist_MapPFB.PantoParE.Macchina.AsseVerticaleY= 0;

Ist_MapPFB.HeaderA.Warn.ParametriLubMancanti:= 	(Ist_MapPFB.PantoParE.Globali.Lub1_enable AND Ist_MapPFB.PantoParE.Macchina.Lub[1].Lub_Lunghezza = 0)
											OR	(Ist_MapPFB.PantoParE.Globali.Lub2_enable AND Ist_MapPFB.PantoParE.Macchina.Lub[2].Lub_Lunghezza = 0);


Ist_MapPFB.HeaderA.Warn.FuoriIngombroInconsistente:= 	Ist_MapPFB.PantoParE.Macchina.ParkZone.AllungMax = 0
												OR	Ist_MapPFB.PantoParE.Macchina.ParkZone.AllungMin = 0;

Ist_MapPFB.HeaderA.Warn.AngleArmsGainMissing:= 	Ist_MapPFB.PantoParE.Sensori.AngoloBraccio.Gain = 0;
Ist_MapPFB.HeaderA.Warn.ZAxisGainMissing:=		Ist_MapPFB.PantoParE.Sensori.Z.Gain = 0;
Ist_MapPFB.HeaderA.Warn.LengthArmsGainMissing:= 	Ist_MapPFB.PantoParE.Sensori.EstBraccio.Gain = 0;
Ist_MapPFB.HeaderA.Warn.NoGainAsseZ2:=			Ist_MapPFB.PantoParE.Sensori.Z2.Gain = 0;
Ist_MapPFB.HeaderA.Warn.NoGainPolso:=			Ist_MapPFB.PantoParE.Sensori.Polso.Gain = 0;
END_FUNCTION_BLOCK

(* POU LifeBit, ST *)
FUNCTION_BLOCK LifeBit
VAR_INPUT
	NumCicli:INT;	(*numero cicli di life bit alzato *)
END_VAR
VAR_OUTPUT
	LifeBit: BOOL;
END_VAR
VAR
	Cicli:	INT;
	resto:	INT;
END_VAR
IF NumCicli<> 0
THEN
	cicli:= cicli +1;
	resto:= cicli MOD (NumCicli*2);
	
	IF resto <= (NumCicli-1)
	THEN
		LifeBit:= TRUE;
	ELSE
		LifeBit:= FALSE;
	END_IF
ELSE
	LifeBit:= FALSE;
END_IF

IF cicli > 1000
THEN
	cicli:=0;
END_IF
END_FUNCTION_BLOCK

(* POU Pantografo/FB_SystemPantoNEW, ST *)
FUNCTION_BLOCK FB_SystemPantoNEW
VAR_INPUT
	L1_Lungh:		REAL;	(**)
	L1_AngleType:	REAL;		(*0: L1 allineato; 90: angolo esterno; -90: angolo interno*)
	Braccio_Est:		REAL;	(*risultato del sensore dell'estensione braccio*)
	Braccio_Rad:		REAL;	(*risultato del sensore dell'angolo braccio*)
	ZBraccio:		REAL;	(*risultato del sensore altezza braccio*)
	ZBraccio2:		REAL;	(*risultato del sensore compensazioneZ; se ZERO non inficia il calcolo*)
	RadPiano:		REAL;	(*risultato del Sensore di rotazione Pallet*)
	Polso_Rad:		REAL;	(*risultato del sensore dell'angolo polso*)
	Chiave1:			Lubbering;
	Chiave2:			Lubbering;
	Lub1_en:			BOOL;	(*Abilitazione Lub1*)
	Lub2_en:			BOOL;	(*Abilitazione Lub1*)
	PianoRot_en:		BOOL;	(*Abilitazione Piano Rotante*)
	X_Offset:			REAL;
	Y_Offset:			REAL;
END_VAR
VAR_OUTPUT
	ActualPosition:	Coordinate;
END_VAR
VAR
	PuntoBraccio:			Coordinate;	(*coordinate dell'estremità del braccio*)
	PuntoLub:			Coordinate; 	(*coordinate sulla chiave Lubbering con origine il punto braccio*)
	Chiave:				Lubbering;	(*chiave in uso*)
	ActualPosition_NoROT:Coordinate;	(*coordinata attuale prima della rotazione del piano*)
	PolarCoord_tmp:		PolarCoord;
	Angolo_K:			REAL;
	(*angolo compensazione disallineamento punto_chiave con asseZ*)

END_VAR
(**********************INIT************************)
IF Lub1_en THEN
	Chiave:=  Chiave1;
END_IF
IF Lub2_en THEN
	Chiave:=  Chiave2;
END_IF



(***calcolo PUNTO BRACCIO******)

IF L1_AngleType=0 THEN
	PuntoBraccio.Angle:= Braccio_Rad;
	PuntoBraccio.Distance:= Braccio_Est;

ELSIF L1_AngleType=90 THEN
	PuntoBraccio.Distance:= SQRT(Braccio_Est*Braccio_Est +L1_Lungh*L1_Lungh);
	Angolo_K:= ASIN(L1_Lungh/PuntoBraccio.Distance);
	PuntoBraccio.Angle:=Braccio_Rad-Angolo_K;
ELSIF L1_AngleType=-90 THEN
	PuntoBraccio.Distance:= SQRT(Braccio_Est*Braccio_Est +L1_Lungh*L1_Lungh);
	Angolo_K:= -ASIN(L1_Lungh/PuntoBraccio.Distance);
	PuntoBraccio.Angle:=Braccio_Rad+Angolo_K;
END_IF

PuntoBraccio.X:= COS(PuntoBraccio.Angle)*PuntoBraccio.Distance + X_Offset;;
PuntoBraccio.Y:= SIN(PuntoBraccio.Angle)*PuntoBraccio.Distance  + Y_Offset;;
PuntoBraccio.Z:= ZBraccio - ZBraccio2;

IF Lub1_en OR Lub2_en THEN
	IF L1_AngleType=0 		THEN 	PuntoLub.Angle:= PuntoBraccio.Angle + Polso_Rad + Chiave.AngoloMontaggio;
	ELSIF L1_AngleType=90 	THEN	PuntoLub.Angle:= PuntoBraccio.Angle + Polso_Rad + Chiave.AngoloMontaggio  - ABS(Angolo_K);
	ELSIF L1_AngleType=-90  	THEN	PuntoLub.Angle:= PuntoBraccio.Angle + Polso_Rad + Chiave.AngoloMontaggio + ABS(Angolo_K);
	END_IF

	PuntoLub.Distance:= Chiave.Lub_Lunghezza;

	PuntoLub.X:= PuntoBraccio.X + COS(PuntoLub.Angle)*PuntoLub.Distance;
	PuntoLub.Y:= PuntoBraccio.Y + SIN(PuntoLub.Angle)*PuntoLub.Distance;
	PuntoLub.Z:= PuntoBraccio.Z;

END_IF

ActualPosition_NoROT := SEL( (Lub1_en OR Lub2_en) , PuntoBraccio, PuntoLub);

IF PianoRot_en
THEN


	(*calcolo coordinata polare rispetto all'origine*)
	PolarCoord_tmp:=FC_CalcRandAngle(	X1:= 0,
										Y1:= 0,
										X2 :=ActualPosition_NoROT.X,
										y2 := ActualPosition_NoROT.Y);

	ActualPosition.Angle:=PolarCoord_tmp.Angle;
	ActualPosition.Distance:=PolarCoord_tmp.Distance;

(*Compensazione con l'angolo di rotazione e calcolo delle nuove coordinate*)
	ActualPosition.X:= COS(PolarCoord_tmp.Angle - RadPiano)*PolarCoord_tmp.Distance;(*+ X_Offset,*)
	ActualPosition.Y:= SIN(PolarCoord_tmp.Angle - RadPiano)*PolarCoord_tmp.Distance;(*+ Y_Offset*)
	ActualPosition.Z:=	ActualPosition_NoROT.Z;

ELSE
	ActualPosition:=	ActualPosition_NoROT;
END_IF
END_FUNCTION_BLOCK

(* POU Pantografo/FC/FC_CalcRandAngle, ST *)
FUNCTION FC_CalcRandAngle : PolarCoord
	(*Calcola Angolo e Distanza tra Punto1 -riferimento-  e Punto 2*)
VAR_INPUT
	X1:	REAL;	(*X1,Y1 coordinate del Punto1 --> per noi sarà l'origine Assi del piano XY che corrisponderà al Centro Portapezzo*)
	Y1:	REAL;
	X2:	REAL;	(*X1,Y1 coordinate del Punto2*)
	Y2:	REAL;
END_VAR
VAR
	DeltaX:		REAL;
	DeltaY:		REAL;
	Segmento:	REAL;
	Angle:		REAL;
END_VAR
VAR CONSTANT
(*messe nelle GLOBALI
	PiGreco: REAL := 3.14159265358979;
	PiGreco2: REAL:= 6.28318530717958;
	PiGrecoMezzi: REAL:= 1.5707963267949;
	PiGreco3Mezzi: REAL:= 4.71238898038469;*)
END_VAR
(*calcolo del segmento tra i punti P1 e P2 --> Teorema di Pitagora*)
DeltaX:= X2 - X1;
DeltaY:=	Y2 - Y1;
Segmento := SQRT((DeltaX * DeltaX) +(DeltaY * DeltaY));

(*Angolo*)
IF DeltaX<>0
THEN
	Angle:= ATAN(ABS( DeltaY / DeltaX ));
	(*verifica del quadrante di appartenenza*)
	IF DeltaX < 0 AND DeltaY >0
	THEN
		Angle:=  PiGreco - Angle;	(*180°-->PiGreco 	90°-->PiGreco/2*)
	
	ELSIF DeltaX < 0 AND DeltaY < 0
	THEN
		Angle:= Angle + PiGreco;
	
	ELSIF DeltaX > 0 AND DeltaY < 0
	THEN
		Angle:= (PiGreco2) - Angle;
	END_IF
ELSIF DeltaY > 0
THEN
	Angle:= 	PiGrecoMezzi;
ELSIF DeltaY < 0
THEN
	Angle:= 	PiGreco3Mezzi;
END_IF

FC_CalcRandAngle.Angle		:= Angle;
FC_CalcRandAngle.Distance	:= Segmento;
END_FUNCTION

(* POU Pantografo/Matching/FB_Std_Match, ST *)
FUNCTION_BLOCK FB_Std_Match
VAR_INPUT
	Actualpoint: 	Coordinate;
	Point2Match:	Coordinate; 			(*punti da matchare - passare la coordinata per ogni vite*)
	R_Toll: 	REAL;					(*raggio di tolleranza del punto da matchare*)
	Z_Toll:	REAL; 					(*Tolleranza "simmetrica" Verticale *)
	Z_Min: 	REAL; 					(*altezza minima Verticale per il controllo a fine avvitatura*)
	Z_Max: 	REAL; 					(*altezza massima Verticale per il controllo a fine avvitatura*)
	ZCheck: 		BOOL;				(*abilitazione controllo di Z: Tolleranza Z per abilitare l'avvitatura*)
	ZCheckFinale:BOOL;				(*controllo finale di Z: altezza min e altezza max dopo l'avvitatura*)
	PianoCheck: 	BOOL;				(*abilitazione del controllo sul piano XY*)
	oscill:		REAL;				(*Valore di Tolleranza di Oscillazione*)
	oscill_Default: REAL;				(*Valore di default della Tolleranza di oscillazione*)
	oscill_Ev:	BOOL;				(*se l'evento è TRUE viene considerato oscill, altrimenti  oscill_Default (si consiglia ZERO)*)
	EsitoAvvitatura:	BYTE;			(*esito avvitatura 0 non effettuata 1 ok 2 scarto*)
END_VAR
VAR_OUTPUT
	AreaLarga_OK:	BOOL;			(*il punto è dentro l'area larga*)
	AreaStretta_OK:	BOOL;			(*il punto è dentro l'area stretta*)
END_VAR
VAR
	(*oscill:		REAL;	(*da toglere son l'FB Std*) per la versione NON STD*)
	deltaX:		REAL;
	deltaY:		REAL;
	deltaR:		REAL;
	(*SR_MatchLargo:	SR;
	SR_MatchStretto:	SR;*)
END_VAR
oscill := SEL(oscill_Ev, oscill_Default, oscill); (*se l'evento è falso viene assume valore oscill_Default*)

deltaX:= actualpoint.X - Point2Match.X;
deltaY:= actualpoint.Y - Point2Match.Y;
deltaR:= SQRT((deltaX*deltaX) + (deltaY*deltaY));

IF (deltaR <= R_Toll + oscill OR NOT PianoCheck)
AND(	( actualpoint.Z >= Point2Match.Z - Z_Toll  AND actualpoint.Z <= Point2Match.Z + Z_Toll )
	OR NOT ZCheck) AND (EsitoAvvitatura <> 1)
THEN
	AreaLarga_OK:= TRUE;
ELSE
	AreaLarga_OK:= FALSE;
END_IF

IF 	(deltaR <= R_Toll + oscill OR NOT PianoCheck)
AND(	(actualpoint.Z >= Z_Min AND actualpoint.Z <= Z_Max)
	OR NOT ZCheckFinale) AND (EsitoAvvitatura <> 1)
THEN
	AreaStretta_OK:= TRUE;
ELSE
	AreaStretta_OK:= FALSE;
END_IF
END_FUNCTION_BLOCK

(* POU Pantografo/FC/FC_InitArea, ST *)
FUNCTION FC_InitArea : ARRAY [1..MaxViti] OF BOOL
VAR_INPUT
	Area:	ARRAY [1..MaxViti] OF BOOL;
END_VAR
VAR
	iArea:	BYTE;
END_VAR
FOR iArea:=1 TO MaxViti
DO
	Area[iArea]:= FALSE;
END_FOR
FC_InitArea:= Area;
END_FUNCTION

(* POU Pantografo/Matching/FC_Avvitabile, ST *)
FUNCTION FC_Avvitabile : BOOL (*FC NON STANDARD ma  legata alla Struct Prodotto*)
VAR_INPUT
	id_avv :	BYTE;	(*id della vite che corrisponde all'indice dell'Array PuntiVite*)
	id_flangia: BYTE;
END_VAR
VAR
END_VAR
VAR CONSTANT
(* nelle Variabili GLOBALI
	Scarto:		BYTE:= 2;
	Good: 		BYTE:= 1;
	NonEffettuata :BYTE := 0;*)
END_VAR
FC_Avvitabile:= 	(Prodotto.PuntoVite[id_flangia,id_avv].EsitoAvvitatura= NonEffettuata)		(*l'avvitatura sul punto non è stata ancora effettuata *)
				OR
                                              (Prodotto.PuntoVite[id_flangia,id_avv].EsitoAvvitatura = Svitare		(* oppure è stata scartata AND abbiamo l'opzione di riavvitabilità*)
					 AND Prodotto.PuntoVite[id_flangia,id_avv].ProgSvitatura <> 0)
				OR
                                              (Prodotto.PuntoVite[id_flangia,id_avv].EsitoAvvitatura = Riavvitare)	(* oppure è stata svitata*)
				OR
                                              (Prodotto.PuntoVite[id_flangia,id_avv].EsitoAvvitatura = NonSvitabile);	(* oppure non può essere svitata *)
END_FUNCTION

(* POU Pantografo/ScrewDataReceiving/FC_PuntoViteAppend, ST *)
FUNCTION FC_PuntoViteAppend : BYTE
VAR_INPUT
END_VAR
VAR
	tmp_IDVite : BYTE;	(*appoggio per index vite*)
	tmp_IDFlangia: BYTE;	(*appoggio per index flangia*)
END_VAR
(* messe nella globali
VAR CONSTANT
	Scarto:		BYTE:= 2;
	Good: 		BYTE:= 1;
	NonEffettuata :BYTE := 0;
END_VAR*)
FC_PuntoViteAppend := NonSvitabile;

tmp_IDVite := Ist_MapPFB.ScrewingE.Id_ViteInviata;  (*appoggio per index vite*)
tmp_IDFlangia:= Ist_MapPFB.ScrewingE.FlangiaInviata;


(*------------------------Riferimenti Punto Vite*)
Prodotto.PuntoVite[tmp_IDFlangia,tmp_IDVite].ID_vite 			:=	tmp_IDVite; (*ASSEGNAZIONE STUPIDA*)
Prodotto.PuntoVite[tmp_IDFlangia,tmp_IDVite].Chiave 			:=	Ist_MapPFB.ScrewingE.ID_Chiave;
Prodotto.PuntoVite[tmp_IDFlangia,tmp_IDVite].ProgAvvitatura 	:=	Ist_MapPFB.ScrewingE.ProgAvvitatura;
Prodotto.PuntoVite[tmp_IDFlangia,tmp_IDVite].ProgRiavvitatura 	:=	Ist_MapPFB.ScrewingE.ProgRiavvitatura;
Prodotto.PuntoVite[tmp_IDFlangia,tmp_IDVite].ProgSvitatura 		:=	Ist_MapPFB.ScrewingE.ProgSvitatura;
(*------------------------coordinate punto vite*)
Prodotto.PuntoVite[tmp_IDFlangia,tmp_IDVite].Posizione.X := 	Ist_MapPFB.ScrewingE.X;
Prodotto.PuntoVite[tmp_IDFlangia,tmp_IDVite].Posizione.Y := Ist_MapPFB.ScrewingE.Y;
Prodotto.PuntoVite[tmp_IDFlangia,tmp_IDVite].Posizione.Z := Ist_MapPFB.ScrewingE.Z;
(*------------------------Tolleranze di Start Avvitatura*)
Prodotto.PuntoVite[tmp_IDFlangia,tmp_IDVite].TolleranzaR := Ist_MapPFB.ScrewingE.TollR;
Prodotto.PuntoVite[tmp_IDFlangia,tmp_IDVite].TolleranzaZ := Ist_MapPFB.ScrewingE.TollZ;
(*------------------------Tolleranze di Check Finale di posizione*)
Prodotto.PuntoVite[tmp_IDFlangia,tmp_IDVite].AltezzaMin :=  Ist_MapPFB.ScrewingE.ZMin;
Prodotto.PuntoVite[tmp_IDFlangia,tmp_IDVite].AltezzaMax :=  Ist_MapPFB.ScrewingE.ZMax;

FC_PuntoViteAppend:= Good;
END_FUNCTION

(* POU Cycles, ST *)
FUNCTION Cycles : BOOL
VAR_INPUT
END_VAR
VAR
END_VAR
(*----------------------------------------------------------Ciclo  di Matching-------------------------------------*)

(*una qualsiasi vite fa partire il ciclo di matching se non sono terminate le viti trovate *)
Ist_CyclesMatching.IN_Cycle.Cm_ON :=		(	Screw[1] OR Screw[2]  OR Screw[3] OR Screw[4]
										OR 	Screw[5] OR Screw[6] OR Screw[7] OR Screw[8]
										OR 	Screw[9] OR Screw[10] OR Screw[11] OR Screw[12]
										OR 	Screw[13] OR Screw[14] OR Screw[15])
								AND NOT Ist_MapPFB.PantoA.AvvitatureTerminate
								AND NOT Ist_MapPFB.HeaderE.Cmd.TxScrewingData;
Ist_CyclesMatching.IN_Cycle.HOLD := FALSE;
Ist_CyclesMatching.IN_Cycle.STEP := FALSE;
Ist_CyclesMatching();

(*non va bene il solo comando perchè nell'ultimo handshake plcmsg e bkhmsg restano uguali, quindi si salterebbe subito allo stato 15*)
Ist_CyclesDataReceiving.IN_Cycle.Cm_ON :=	Ist_MapPFB.HeaderE.Cmd.TxScrewingData;
Ist_CyclesDataReceiving.IN_Cycle.HOLD := FALSE;
Ist_CyclesDataReceiving.IN_Cycle.STEP := FALSE;
Ist_CyclesDataReceiving();
END_FUNCTION

(* POU Pantografo/ScrewDataReceiving/CyclesDataReceiving, ST *)
FUNCTION_BLOCK CyclesDataReceiving (*struttura: 	Stato <10> :  Inizio HandShake - Lettura del PlcMsgNum ed invio Msg +1
												Stato <15> : Attesa PLCMsg per entrare nello stato di dati affidabili
												Stato <20> : Fase di Accodamento e inizio Handshake2
												Stato <30> :FineHandshake2*)
VAR_INPUT
	IN_Cycle:InputCiclo;
END_VAR
VAR_OUTPUT
	OUT_Cycle:OutputCiclo;
END_VAR
VAR
	Stato:INT;
	StatoSeguente:INT;
	FrontePassoSingolo:BOOL;
	CicloTermOK:BOOL;
	CicloTermKO:BOOL;
	CicloInCorso:BOOL;
	Ist_R_TRIG:R_TRIG;
END_VAR
(*----------------------------------------aggiornamento stato*)
Ist_R_TRIG(CLK:=FrontePassoSingolo);
IF 	(IN_Cycle.STEP AND
	Ist_R_TRIG.Q) OR
	NOT IN_Cycle.HOLD
THEN
	Stato := StatoSeguente;
END_IF

(*-------------------------------------------stati particolari*)
CicloInCorso := Stato <> 0;
CicloTermOK := Stato = 60;
CicloTermKO := Stato = 59;

(*Stato <0> : Ciclo off*)
IF	Stato = 0
THEN
	(*Ist_MapPFB.HeaderA.Com.BeckMsgNum:= 0; (*0 ad inizio e a fine ciclo*)*)
	IF 	IN_Cycle.Cm_ON
	THEN
		StatoSeguente := 10;
	END_IF
END_IF

(*Stato <10> : Inizio HandShake - Lettura del PlcMsgNum ed invio Msg +1 *)
IF 	Stato = 10
THEN	(*prerequisito dell'handshaking*)
	IF Ist_MapPfb.HeaderA.Com.BeckMsgNum = Ist_MapPFB.HeaderE.Com.PlcMsgNum (*OLD  Ist_ToolMapA.BkhMsgNum  = Ist_ToolMapE.PlcMsgNum*)
	THEN
                  Ist_MapPfb.HeaderA.Com.BeckMsgNum := Ist_MapPFB.HeaderE.Com.PlcMsgNum + 1;
		StatoSeguente := 15;
	END_IF
END_IF

(*Stato <15> : Attesa PLCMsg per entrare nello stato di dati affidabili *)
IF 	Stato = 15
THEN
	IF Ist_MapPfb.HeaderA.Com.BeckMsgNum = Ist_MapPFB.HeaderE.Com.PlcMsgNum
	THEN
		StatoSeguente := 20;
	END_IF
END_IF


(*Stati <20> : Stato di Dati Affidabili Attesa fine di Accodamento e inizio Handshake2*)
IF Stato = 20
THEN
	IF Ist_MapPFB.EsitoAccodamento = 1 OR Ist_MapPFB.EsitoAccodamento = 2
	THEN
		StatoSeguente := 30;
		 Ist_MapPfb.HeaderA.Com.BeckMsgNum := Ist_MapPFB.HeaderE.Com.PlcMsgNum + 1;;
	END_IF
END_IF

(*Stato <30> :FineHandshake2*)
IF Stato = 30
THEN
	IF  Ist_MapPFB.HeaderE.Com.PlcMsgNum = Ist_MapPFB.HeaderA.Com.BeckMsgNum (*OLD Ist_ToolMapE.PlcMsgNum =  Ist_ToolMapA.BkhMsgNum*)
	THEN
		StatoSeguente := 60;
	END_IF
END_IF

(*Stato <60> : Fine ciclo OK*)
IF 	NOT IN_Cycle.Cm_ON
THEN
	StatoSeguente := 0;
END_IF

(*Stato <59> : Fine ciclo KO*)
(*IF 	Stato = 59 OR
	NOT IN_Cycle.Cm_ON
THEN
	StatoSeguente := 0;
END_IF*)

(*Uscite*)
OUT_Cycle.Stato := Stato;
OUT_Cycle.CicloInCorso := CicloInCorso;
OUT_Cycle.CicloTerminatoOK := CicloTermOK;
OUT_Cycle.CicloTerminatoKO := CicloTermKO;
END_FUNCTION_BLOCK

(* POU Pantografo/Matching/CyclesMatching, ST *)
FUNCTION_BLOCK CyclesMatching
VAR_INPUT
	IN_Cycle:InputCiclo;
END_VAR
VAR_OUTPUT
	OUT_Cycle:OutputCiclo;
END_VAR
VAR
	Stato:INT;
	StatoSeguente:INT;
	FrontePassoSingolo:BOOL;
	CicloTermOK:BOOL;
	CicloTermKO:BOOL;
	CicloInCorso:BOOL;
	Ist_R_TRIG:R_TRIG;
END_VAR
(*----------------------------------------aggiornamento stato*)
Ist_R_TRIG(CLK:=FrontePassoSingolo);
IF 	(IN_Cycle.STEP AND
	Ist_R_TRIG.Q) OR
	NOT IN_Cycle.HOLD
THEN
	Stato := StatoSeguente;
END_IF

(*-------------------------------------------stati particolari*)
CicloInCorso := Stato <> 0;
CicloTermOK := Stato = 60;
CicloTermKO := Stato = 59;

(*Stato <0> : Ciclo off*)
IF	Stato = 0
THEN
	IF 	IN_Cycle.Cm_ON
	THEN
		StatoSeguente := 5;(*10;*)
	END_IF
END_IF
(*test per vedere avvitatura in corso giu*)
IF	Stato = 5
THEN
	IF NOT  Ist_MapPFB.PantoE.Avvitatura_InCorso
	THEN
		StatoSeguente := 10;
	END_IF
END_IF


(*Stato <10> : StartAvvitatura /avvitatura in corso per avere la certezza che avvitatura fine sia a zero*)
IF 	Stato = 10
THEN
	IF NOT Ist_MapPFB.PantoE.Avvitatura_Fine
	THEN
		 IF Ist_MapPFB.HeaderE.Cmd.Matching
		THEN
			IF NOT Ist_MapPFB.PantoA.AbilitaSvitatura
			THEN
				IF Ist_MapPFB.PantoE.Avvitatura_InCorso
				THEN
					StatoSeguente := 15;
				END_IF
			ELSE
				StatoSeguente :=44;(* 45;*)
			END_IF (*fine controllo di abilita svitatura*)
		END_IF (*fine controllo matching abilitato *)
	END_IF
END_IF

(*Stato <15> : StartAvvitatura / attesa fine avvitatura e Valutazione Esito Avvitatura*)
IF 	Stato = 15
THEN

	IF  Ist_MapPFB.PantoE.Avvitatore_EsitoOK AND Ist_MapPFB.PantoE.Avvitatura_Fine
	THEN
		StatoSeguente := 30;
	END_IF

	IF Ist_MapPFB.PantoE.Avvitatore_EsitoKO AND Ist_MapPFB.PantoE.Avvitatura_Fine
	THEN
		StatoSeguente := 44;
	END_IF
END_IF



(*Stato <30> CheckFinalPosition - Attesa ACK della posizione Finale*)
IF 	Stato = 30
THEN (*nello stato 30 systems attende il match stretto che genera il final position OK*)
	IF Ist_MapPFB.PantoA.Final_Position_OK AND (NOT Ist_MapE.StartPls OR NOT Ist_MapPFB.PantoParE.Globali.ScrewSequenceActive) (*AND Ist_MapPFB.HeaderE.Com.Plc_ACK*)
	THEN
		StatoSeguente := 60;
	END_IF
	IF Ist_MapPFB.PantoA.Final_Position_KO AND (NOT Ist_MapE.StartPls OR NOT Ist_MapPFB.PantoParE.Globali.ScrewSequenceActive)  (*AND Ist_MapPFB.HeaderE.Com.Plc_ACK*)
	THEN
		StatoSeguente :=  44;
	END_IF
END_IF


(*Stato <44> : Attendo il rilascio del pulsante di avvitatura in caso di scarto*)
IF 	Stato = 44
THEN
	IF NOT Ist_MapE.StartPls
	THEN
		StatoSeguente := 45;
	END_IF
END_IF

(*Stato <45> :  Svitatura comandata - Attesa Avvitatura In Corso*)
IF 	Stato = 45
THEN
	 IF NOT Ist_MapPFB.HeaderE.Cmd.Matching OR Ist_MapPFB.PantoE.Avvitatura_Ripeti
	THEN
		StatoSeguente := 10;		(*Se perdo la vite disattivo la svitatura e cerco un nuovo matching  *)
	ELSIF  Ist_MapPFB.PantoE.Avvitatura_InCorso (*OR NOT Ist_MapPFB.PantoParE.Globali.SvitaturaSuScarto*) (*Ist_MapPFB.HeaderE.Com.Plc_ACK*)
	THEN
		StatoSeguente := 50;
	END_IF
END_IF

(*Stato <50> : Attesa Fine Svitatura (ACK)*)
IF 	Stato = 50
THEN
	IF  Ist_MapPFB.PantoE.Avvitatura_Fine OR NOT Ist_MapPFB.PantoE.Avvitatura_InCorso (*OR NOT Ist_MapPFB.PantoParE.Globali.SvitaturaSuScarto*) (*EX  -> st_MapPFB.HeaderE.Com.Plc_ACK*)	THEN
		StatoSeguente := 55;
	END_IF
END_IF


(*Stato <55> : Svitatura Terminata*)
IF 	Stato = 55
THEN
	IF NOT Ist_MapE.StartPls THEN
		StatoSeguente := 59;
	END_IF
END_IF


(*Stato <60> : Fine ciclo OK*)
IF 	Stato = 60 OR
	NOT IN_Cycle.Cm_ON
THEN
	StatoSeguente := 0;
END_IF

(*Stato <59> : Fine ciclo KO*)
IF 	Stato = 59 OR
	NOT IN_Cycle.Cm_ON
THEN
	StatoSeguente := 0;
END_IF

(*Uscite*)
OUT_Cycle.Stato := Stato;
OUT_Cycle.CicloInCorso := CicloInCorso;
OUT_Cycle.CicloTerminatoOK := CicloTermOK;
OUT_Cycle.CicloTerminatoKO := CicloTermKO;
END_FUNCTION_BLOCK

(* POU SiemensConversion/FC_SiemensDWORD, ST *)
FUNCTION FC_SiemensDWORD : DWORD
VAR_INPUT
	DWORD1:	DWORD;
END_VAR
VAR
	word1:WORD;
	word2:WORD;
	word1_swap:WORD;
	word2_swap:WORD;
	DW_Appoggio: DWORD;
END_VAR
DW_Appoggio:= %MD0;	(*backup Dword0*)
%MD0:=DWORD1;
word1:=%MW0;
word2:=%MW2;
(*rotazione*)
word1_swap:= ROL (word1, 8);
word2_swap:= ROL (word2, 8);
(*appoggio delle word sui merker*)
%MW0:=word1_swap;
%MW2:=word2_swap;
(*restituzione DW con i singoli byte invertiti*)
FC_SiemensDWORD:= %MD0;
(*ripristino backup della %MD0 originale*)
%MD0:=DW_Appoggio;
END_FUNCTION

(* POU SiemensConversion/FC_SiemensREAL, ST *)
FUNCTION FC_SiemensREAL : REAL
VAR_INPUT
	DWORD1:	DWORD;
END_VAR
VAR
	word1:WORD;
	word2:WORD;
	word1_swap:WORD;
	word2_swap:WORD;
	DW_Appoggio: DWORD;
	(*per ora utilizziamo puntatore a REAL*)
	tmp_pt_REAL: POINTER TO REAL;
END_VAR
DW_Appoggio:= %MD0;	(*backup Dword0*)

(*appoggio della DWORD dul Merker %MD0*)
%MD0:=DWORD1;
(*prelievo delle 2 singole word*)
word1:=%MW0;
word2:=%MW2;
(*rotazione delle 2 word*)
word1_swap:= ROL (word1, 8);
word2_swap:= ROL (word2, 8);

(*appoggio delle word ruotate sui relativi merker*)
%MW0:=word1_swap;
%MW2:=word2_swap;
(*utilizzo del puntatore a REAL per riassegnare la struttura al tipo real*)
tmp_pt_REAL:= ADR(%MD0);
(*restituzione REAL con i singoli byte invertiti*)
FC_SiemensREAL:= tmp_pt_REAL^;

(*ripristino backup della %MD0 originale*)
%MD0:=DW_Appoggio;
END_FUNCTION

(* POU SiemensConversion/FC_SiemensReal2Dword, ST *)
FUNCTION FC_SiemensReal2Dword : DWORD
VAR_INPUT
	reale1:	REAL;
END_VAR
VAR
	pt_dword: POINTER TO DWORD;
	word1:WORD;
	word2:WORD;
	word1_swap:WORD;
	word2_swap:WORD;
	DW_Appoggio: DWORD;
END_VAR
DW_Appoggio:= %MD0;	(*backup Dword0*)

(*puntatore a dword del reale passato*)
pt_dword:= ADR(reale1);

(*appoggio della DWORD dul Merker %MD0*)
%MD0:=pt_dword^;
(*prelievo delle 2 singole word*)
word1:=%MW0;
word2:=%MW2;
(*rotazione delle 2 word*)
word1_swap:= ROL (word1, 8);
word2_swap:= ROL (word2, 8);

(*appoggio delle word ruotate sui relativi merker*)
%MW0:=word1_swap;
%MW2:=word2_swap;

(*restituzione MD0  con i singoli byte invertiti*)
FC_SiemensReal2Dword:=%MD0;

(*ripristino backup della %MD0 originale*)
%MD0:=DW_Appoggio;
END_FUNCTION

(* POU SiemensConversion/FC_SiemensWORD, ST *)
FUNCTION FC_SiemensWORD : WORD (*scambia byte0 con byte1*)
VAR_INPUT
	word1:	WORD;
END_VAR
VAR
END_VAR
FC_SiemensWORD:= ROL (word1,8);
END_FUNCTION

(* POU Map/MapA, ST *)
FUNCTION_BLOCK MapA
VAR_INPUT
	Frizione			 :	BOOL;
END_VAR
VAR_OUTPUT
END_VAR
VAR
	StartPls:			BOOL;	(*non deve essere scritto dall'esterno scrivibile*)
END_VAR
%QX140.0:= 	 Ist_MapE.StartPls;
Ist_MapPFB.PantoA.FrizioneComandata:= %QX140.0; (*link dello stato frizione comandata*)
%QX0.0:= Ist_MapE.StartPls;
%QX0.1:= Ist_MapE.StartPls;
%QX0.2:= Ist_MapE.StartPls;
%QX0.3:= Ist_MapE.StartPls;
END_FUNCTION_BLOCK

(* POU Map/MapE, ST *)
FUNCTION_BLOCK MapE (*struttura: StartPls dato dall'esterno
								 Angolo Braccio -> 	CH0
								Altezza Z->			CH1
								Estensione Braccio->	CH2
								Angolo Polso->		CH3
								Altezza Z2->			CH3*)
VAR_INPUT
END_VAR
VAR_OUTPUT
(*--------------------SENSORI-------------*)
	RadBraccio:	REAL;
	GradBraccio: REAL;
	Z:			REAL;
	EstBraccio:	REAL;
	RadPolso:	REAL;
	GradPolso:	REAL;
	Z_Braccio2:	REAL;
	StartPls: 		BOOL;	(*pulsante di start avvitatore*)
(*--------------Fine --SENSORI-------------*)
END_VAR
VAR
(*LOCALI per la linearizzazione dei sensori*)
	(*--------------ANGOLO BRACCIO-------------*)
	RadBraccio_W:	WORD;		(*mappare ai realivi ingressi AT %IWxx *)
	RadBraccio_Gain:			REAL;
	RadBraccio_GainRecipe:	REAL;
	RadBraccio_Offset: 		REAL;
	RadBraccio_OffsetRecipe: 	REAL;
	RadBraccio_LinkedOffset:	REAL; (*l'angolo di montaggio del sensore - offset montaggio*)
	RadBraccio_LinkedGain:	REAL;
	RadBraccio_tmp:	REAL;
	(*--------------ALTEZZA  BRACCIO-------------*)
	Z_W:			WORD;
	Z_Gain:			REAL;
	Z_Offset:			REAL;
	Z_Gain_Recipe:	REAL;
	Z_Offset_Recipe:	REAL;
	Z_LinkedGain:	REAL;
	Z_LinkedOffset:	REAL;
	(*--------------ESTENSIONE BRACCIO----------*)
	EstBraccio_W:	WORD;
	EB_Gain: 	REAL;
	EB_Offset:		REAL;
	EB_Gain_Recipe:	REAL;
	EB_Offset_Recipe:REAL;
	EB_LinkedGain:	REAL;	(*EstBraccio Linear Gain*)
	EB_LinkedOffset:	REAL;	(*EstBraccio Linear Gain*)
	(*--------------ANGOLO POLSO-------------*)
	RadPolso_W:			WORD;
	RadPolso_Gain:			REAL;
	RadPolso_Offset: 			REAL;
	RadPolso_Gain_Recipe:	REAL;
	RadPolso_Offset_Recipe:	REAL;
	RadPolso_LinkedGain: 	REAL;
	RadPolso_LinkedOffset: 	REAL;
	RadPolso_tmp:			REAL;

	(*--------------ANGOLO BRACCIO2 - COMPENSAZIONE DI ----------*)
	Z2_W:			WORD;
	Z2_Gain:			REAL;
	Z2_Offset:		REAL;
	Z2_GainRecipe:	REAL;
	Z2_OffsetRecipe:	REAL;
	Z2_LinkedGain:	REAL;
	Z2_LinkedOffset:	REAL;
	(*Rad_Pallet_W:	WORD;*)
END_VAR
VAR CONSTANT
(*messe nelle GLOBALI
	PiGreco: 			REAL := 3.14159265358979;					(*180 gradi*)
	PiGreco2: 		REAL:= 6.28318530717958;					(*360 gradi*)
	PiGrecoMezzi: 	REAL:= 1.5707963267949;					(*90 gradi*)
	PiGreco3Mezzi: 	REAL:= 4.71238898038469;					(*270 gradi*)
	Pigreco4i: 		REAL := 0.78539816339744830961566084581988;				(*45 gradi*)
	Pigreco3_8:		REAL:= 1.1780972450961724644234912687298;	(*60 gradi*)
	Rad2Gr:			REAL:= 57.295779513082320876798154814105; (*coeff. di conversione: 360 / (2*Pigreco)*)*)
END_VAR
StartPls := %IX8.0;(*Ist_MapPFB.PantoE.StartPls;  dato dal partner profibus esterno*)


(*------------Sensore Angolo Braccio in radianti-----------*)
	RadBraccio_W:= 			%IW0;(*complex%IW2;*)(*%IW0;*)			(*indirizzo fisico -> misura sensore inversa*)
	RadBraccio_LinkedOffset:=	90.0; 	(*in gradi*)
	RadBraccio_LinkedGain:=	Pigreco2/32767;
	RadBraccio_OffsetRecipe:= Ist_MapPFB.PantoParE.Sensori.AngoloBraccio.Offset;	(*mapping alla rete profibus*)
	RadBraccio_GainRecipe:=	Ist_MapPFB.PantoParE.Sensori.AngoloBraccio.Gain;
	(*se il valore dalla rete manca uso il gain e l'offset linkati sul sw in fase di messa in servizio*)
	RadBraccio_Offset:= 		SEL (RadBraccio_OffsetRecipe=0, RadBraccio_OffsetRecipe/ Rad2Gr , RadBraccio_LinkedOffset/ Rad2Gr);
	RadBraccio_Gain:= 		SEL (RadBraccio_GainRecipe= 0, RadBraccio_GainRecipe, RadBraccio_LinkedGain);
	RadBraccio_tmp:= 		(WORD_TO_REAL(RadBraccio_W) * RadBraccio_Gain) + RadBraccio_Offset;

	RadBraccio:= 			SEL (RadBraccio_tmp > Pigreco2, RadBraccio_tmp, RadBraccio_tmp - PiGreco2);	(*se supera 360° tolgo 360°*)

	GradBraccio:= RadBraccio * Rad2Gr;

(*------------Sensore Altezza Z-----------*)
	Z_W:= 			%IW2;(*complex%IW6;*)(*%IW2;*)			(*indirizzo fisico-> misurazione invertita*)
	Z_Gain_Recipe:=	Ist_MapPFB.PantoParE.Sensori.Z.Gain;		(*mapping alla rete profibus*)
	Z_Offset_Recipe:=	Ist_MapPFB.PantoParE.Sensori.Z.Offset;
	Z_LinkedGain:=	0.0148957298907646; 	(*rapporto Delta Z mm/DeltaWORD -> DA FARE*)
	Z_LinkedOffset:= 	0.0;
	Z_Gain:= 		SEL (Z_Gain_Recipe= 0, Z_Gain_Recipe , Z_LinkedGain);

	Z_Offset:=		SEL(Z_Offset_Recipe= 0, Z_Offset_Recipe, Z_LinkedOffset);
						(* misurazione invertita*)
	Z:=  (WORD_TO_REAL(32767 - Z_W) * Z_Gain) +Z_Offset;

(*------------Sensore Estensione Braccio-----------*)
	EstBraccio_W:= 		%IW4;(*copmlex%IW10;*)(*%IW4;*)			(*indirizzo fisico*)
	EB_Gain_Recipe:=	Ist_MapPFB.PantoParE.Sensori.EstBraccio.Gain;		(*mapping alla rete profibus*)
	EB_Offset_Recipe:=	Ist_MapPFB.PantoParE.Sensori.EstBraccio.Offset;
	EB_LinkedGain:=		-0.0147227533460803; 	(*rapporto Delta  mm/DeltaWORD -> DA FARE*)
	EB_LinkedOffset:=		709.0;
	EB_Gain:= 			SEL (EB_Gain_Recipe= 0, EB_Gain_Recipe , EB_LinkedGain);
	EB_Offset:=			SEL(EB_Offset_Recipe= 0, EB_Offset_Recipe, EB_LinkedOffset);

	EstBraccio:=  			 (WORD_TO_REAL(EstBraccio_W) * EB_Gain) +EB_Offset;

(*------------Sensore Angolo Polso in radianti-----------*)
	RadPolso_W:= 			%IW6;(*copmlex%IW12;*)(*%IW6;*)			(*indirizzo fisico*)
	RadPolso_LinkedOffset:=	141.34; 	(*in gradi*)
	RadPolso_LinkedGain:=	Pigreco2/32767;
	RadPolso_Offset_Recipe:= Ist_MapPFB.PantoParE.Sensori.Polso.Offset;	(*mapping alla rete profibus*)
	RadPolso_Gain_Recipe:=	Ist_MapPFB.PantoParE.Sensori.Polso.Gain;
	(*se il valore dalla rete manca uso il gain e l'offset linkati sul sw in fase di messa in servizio*)
	RadPolso_Offset:= 	SEL (RadPolso_Offset_Recipe=0, RadPolso_Offset_Recipe/ Rad2Gr , RadPolso_LinkedOffset/ Rad2Gr);
	RadPolso_Gain:= 		SEL (RadPolso_Gain_Recipe= 0, RadPolso_Gain_Recipe, RadPolso_LinkedGain);
	RadPolso_tmp:= 		(WORD_TO_REAL(RadPolso_W) * RadPolso_Gain) + RadPolso_Offset;

	IF RadPolso_tmp < 0
	THEN
		RadPolso:= 			RadPolso_tmp+PiGreco2;
	ELSIF RadPolso_tmp > PiGreco2
		THEN
		RadPolso:= 			RadPolso_tmp-PiGreco2;
	ELSE
			RadPolso:=		RadPolso_tmp;
	END_IF




(*SEL (RadPolso_tmp > Pigreco2, RadPolso_tmp, RadPolso_tmp - PiGreco2);	(*se supera 360° tolgo 360°*)*)

	GradPolso:= RadPolso * Rad2Gr;

(*------------Sensore Altezza Z2-----------*)
IF Ist_MapPFB.PantoParE.Globali.Lub1_enable OR Ist_MapPFB.PantoParE.Globali.Lub2_enable
THEN
	Z_Braccio2:= 0;
ELSE
	Z2_W:= 			%IW6;			(*indirizzo fisico*)
	Z2_GainRecipe:=	Ist_MapPFB.PantoParE.Sensori.Z2.Gain;		(*mapping alla rete profibus*)
	Z2_OffsetRecipe:=	Ist_MapPFB.PantoParE.Sensori.Z2.Offset;
	Z2_LinkedGain:=	0.000477962514082824; 	(*rapporto Delta Z mm/DeltaWORD -> DA FARE*)
	Z2_LinkedOffset:= 	-1.255606;
	Z2_Gain:= 		SEL (Z2_GainRecipe= 0, Z2_GainRecipe , Z2_LinkedGain);

	Z2_Offset:=		SEL(Z2_OffsetRecipe= 0, Z2_OffsetRecipe, Z2_LinkedOffset);

	Z_Braccio2:=  	(WORD_TO_REAL(Z2_W) * Z2_Gain) +Z2_Offset;
END_IF
END_FUNCTION_BLOCK

(* POU Map/MapPFB, ST *)
FUNCTION_BLOCK MapPFB(*struttura: 	Header E	->	COMUNICAZIONE - LIFE BIT
												->	COMANDI
												->	WARNING
									Header A	->	COMUNICAZIONE
												->	ECHO COMANDI
												->	WARNING
									MapPantoE
									MapPantoParE ->	GLOBALI
												->	MACHINE
												->	SENSORI
									MapPantoA	
									MapPantoParA->	GLOBALI
												->	MACHINE
												->	SENSORI
									Re-link ECHO
									TxScrewing*)
VAR_INPUT
(*istanze comuni*)
	HeaderA:	MapHeaderA;
(*istanze di Pantorafo Enable*)
	(*uscite di Pantografo Enable*)
	PantoA:		MapPantoA;
	(*PantoParA:	MapPantoParA;*)
	EsitoAccodamento:	BYTE;
END_VAR
VAR_OUTPUT
(*istanze comuni*)
	HeaderE:	MapHeaderE;
(*istanze di Pantografo Enable*)
	(*ingressi di Pantografo Enable*)
	PantoE:		MapPantoE;
	PantoParE:	MapPantoParE;
	(*ingressi di TxScrewingData*)
	ScrewingE:		MapScrewingE;
END_VAR
VAR
END_VAR
(*---------Mapping su PFB Header E ---------*)
	(*COMUNICAZIONE - LIFE BIT*)
HeaderE.Com.PlcMsgNum:=	%IB128;
HeaderE.Com.PlcLifeBit:= 		%IX129.0;
HeaderE.Com.EchoBeckBit:=	%IX129.1;
HeaderE.Com.Plc_ACK:=		%IX129.2;

	(*COMANDI*)
HeaderE.Cmd.Matching:= 				%IX130.0;
HeaderE.Cmd.TxScrewingData:=		%IX130.1;
HeaderE.Cmd.RqstScrewingData:=		%IX130.2;
HeaderE.Cmd.ResettaEsitiAvvitature:=	%IX130.3	;

(* not used
	(*WARNING*)
HeaderE.WarnECHO.RicettaVuota:= 				%IX132.0;
HeaderE.WarnECHO.OffsetMancante:= 			%IX132.1;
HeaderE.WarnECHO.ParametriLubMancanti:= 		%IX132.2;
HeaderE.WarnECHO.FuoriIngombroInconsistente:= %IX132.3;
HeaderE.WarnECHO.AngleArmsGainMissing:= 	%IX132.4;
HeaderE.WarnECHO.ZAxisGainMissing:= 			%IX132.5;
HeaderE.WarnECHO.LengthArmsGainMissing:= 	%IX132.6;
HeaderE.WarnECHO.NoGainAsseZ2:= 			%IX132.7;
HeaderE.WarnECHO.NoGainPolso:= 			%IX132.7; (*si userà Z2 oppure il polso*)
*)

(*---------Mapping su PFB Header A ---------*)
	(*COMUNICAZIONE*)
(*%QW128:= 0;	(*OUT inizializzazione dei 16 bit di comunicazione*)*)

%QB128:= 	HeaderA.Com.BeckMsgNum;
%QX129.0:=	HeaderA.Com.EchoPLCLifeBit;
%QX129.1:=	HeaderA.Com.BeckLifeBit;
%QX129.2:=	HeaderA.Com.Beck_ACK;

	(*ECHO COMANDI - not used*)
(*%QW130:= 0; (*OUT inizializzazione dei 16 bit di comandi - 8MacroCom + 8 Comandi*)*)
(*not used
%QX130.0:= 	HeaderA.CmdECHO.Matching;
%QX130.1:= 	HeaderA.CmdECHO.TxScrewingData;
%QX130.2:= 	HeaderA.CmdECHO.RqstScrewingData;
*)

	(*WARNING*)
(*%QW132:= 	0;	(*inizializzazione allarmi*)*)
%QX132.0:=	HeaderA.Warn.RicettaVuota;
%QX132.1:=	HeaderA.Warn.OffsetMancante;
%QX132.2:=	HeaderA.Warn.ParametriLubMancanti;
%QX132.3:=	HeaderA.Warn.FuoriIngombroInconsistente;
%QX132.4:=	HeaderA.Warn.AngleArmsGainMissing;
%QX132.5:=	HeaderA.Warn.ZAxisGainMissing;
%QX132.6:=	HeaderA.Warn.LengthArmsGainMissing;
%QX132.7:=	HeaderA.Warn.NoGainAsseZ2 OR HeaderA.Warn.NoGainPolso;
(*Alarms %QX134.0 .. %QX135.7*)

(*MacroStati %QX136.0..%QX137.7*)
(*%QX136.0:= Pantografo Enabled non usato*)
%QX136.1:= HeaderA.MacroStati.TxScrewingData;
(*%QX136.2 non usato*)
%QX136.3:=HeaderA.MacroStati.EsitiavvitatureResettati;



(*-----------------Mapping su PFB MapPantoE----------*)
(*PantoE.StartPls:=				%IX140.0;*)
PantoE.Avvitatore_EsitoOK:= 	%IX140.2;
PantoE.Avvitatore_EsitoKO:= 	%IX140.3;
PantoE.Avvitatura_InCorso:= 	%IX140.4;
PantoE.Avvitatura_Fine:= 		%IX140.5;
PantoE.Avvitatura_Ripeti:=		%IX140.6;
PantoE.ECHO_Viti_Effettuate:= 	%IB141;	(*attenzione  viene rimappato come Id_vite inviata in caso di Ricezione avvitatura*)
PantoE.Viti_Totali_Flangia:=	%IB142;
PantoE.FlangiaInCorso:=		%IB143;
PantoE.AngoloPallet:=	FC_SiemensREAL(DWORD1:=%ID144);
PantoE.ProgAvvitGenerico:=	%IB148;


(*mapping del pantografo -> quando il PLC non invia nè richiede i punti vite VALUTARE SE SERVE O MENO INTERBLOCCARE il mapping di ingresso *)
IF 	NOT HeaderE.Cmd.TxScrewingData
	AND NOT HeaderE.Cmd.RqstScrewingData
THEN
(*-------------mapping su PFB MapPantoParE-------------*)
	(*GLOBALI*)
	PantoParE.Globali.ProgrammaSvitatura:= 		%IB156;
	PantoParE.Globali.SvitaturaSuScarto:= 		%IX157.0;
	PantoParE.Globali.CheckZ:=				%IX157.1;
	PantoParE.Globali.CheckPianoXY:=			%IX157.2;
	PantoParE.Globali.CheckZfinale:=			%IX157.3;
	PantoParE.Globali.PianoRotanteAttivo:=		%IX157.4;
	PantoParE.Globali.Lub1_enable:=			%IX157.5;
	PantoParE.Globali.Lub2_enable:=			%IX157.6;
	PantoParE.Globali.ScrewSequenceActive:=	%IX157.7;
	(*MACHINE*)

	PantoParE.Macchina.AsseVerticaleX:= 	FC_SiemensREAL(DWORD1:=%ID158);
	PantoParE.Macchina.AsseVerticaleY:= 	FC_SiemensREAL(DWORD1:=%ID162);
	PantoParE.Macchina.L1_lunghezza:= 		FC_SiemensREAL(DWORD1:=%ID166);
	PantoParE.Macchina.L1_Angolo:= 		FC_SiemensREAL(DWORD1:=%ID170);
	PantoParE.Macchina.OscillAvvitatore:= 	FC_SiemensREAL(DWORD1:=%ID174);

	(*-----------SEZIONE CHIAVI-------------------*)
		(*-------------chiave 1----------------*)
	PantoParE.Macchina.Lub[1].AngoloMontaggio:=	FC_SiemensREAL(DWORD1:=%ID178);
	PantoParE.Macchina.Lub[1].Lub_Lunghezza:=		FC_SiemensREAL(DWORD1:=%ID182);
		(*-------------chiave 2----------------*)
	PantoParE.Macchina.Lub[2].AngoloMontaggio:=	FC_SiemensREAL(DWORD1:=%ID186);
	PantoParE.Macchina.Lub[2].Lub_Lunghezza:=		FC_SiemensREAL(DWORD1:=%ID190);

	(*-----------SEZIONE PARKING ZONE-------------------*)
	PantoParE.Macchina.ParkZone.AllungMax:=	FC_SiemensREAL(DWORD1:=%ID194);
	PantoParE.Macchina.ParkZone.AllungMin:=	FC_SiemensREAL(DWORD1:=%ID198);
	PantoParE.Macchina.ParkZone.AngoloMax:=	FC_SiemensREAL(DWORD1:=%ID202);
	PantoParE.Macchina.ParkZone.AngoloMin:=	FC_SiemensREAL(DWORD1:=%ID206);
	PantoParE.Macchina.ParkZone.AltezzaMin:=	FC_SiemensREAL(DWORD1:=%ID210);
	(*SENSORI*)
	PantoParE.Sensori.AngoloBraccio.Gain := 	FC_SiemensREAL(DWORD1:=%ID214);
	PantoParE.Sensori.AngoloBraccio.Offset := 	FC_SiemensREAL(DWORD1:=%ID218);
	PantoParE.Sensori.Z.Gain := 				FC_SiemensREAL(DWORD1:=%ID222);
	PantoParE.Sensori.Z.Offset := 				FC_SiemensREAL(DWORD1:=%ID226);
	PantoParE.Sensori.EstBraccio.Gain := 		FC_SiemensREAL(DWORD1:=%ID230);
	PantoParE.Sensori.EstBraccio.Offset := 		FC_SiemensREAL(DWORD1:=%ID234);
	(*a seconda della configurazione allo stesso indirizzo c'è l'uno o l'altro*)
	PantoParE.Sensori.Z2.Gain := 		FC_SiemensREAL(DWORD1:=%ID238);
	PantoParE.Sensori.Z2.Offset := 		FC_SiemensREAL(DWORD1:=%ID242);
						(**)
	PantoParE.Sensori.Polso.Gain := 	FC_SiemensREAL(DWORD1:=%ID246);
	PantoParE.Sensori.Polso.Offset := 	FC_SiemensREAL(DWORD1:=%ID250);



END_IF
(*-------------mapping su PFB MapPantoA-------------*)
%QX140.0:= 	PantoA.FrizioneComandata;
%QX140.1:= 	PantoA.ParkingPosition; (*ha senso se non c'è il relativo WARNING*)
%QX140.2:= 	PantoA.AbilitaAvvitatura;
%QX140.3:= 	PantoA.AbilitaSvitatura;
%QX140.4:= 	PantoA.Final_Position_OK;
%QX140.5:= 	PantoA.Final_Position_KO;
%QX140.6:= 	PantoA.AvvitatureTerminate;
%QX140.7:=	PantoA.FrizioneComandata;
%QB141:=	PantoA.Vite_in_Corso;
%QB142:=	PantoA.ProgAvvitatura;
%QB143:=	PantoA.VitiEffettuate;
%QD144:=	FC_SiemensReal2Dword(reale1:=PantoA.X) ;
%QD148:=	FC_SiemensReal2Dword(reale1:=PantoA.Y) ;
%QD152:=	FC_SiemensReal2Dword(reale1:=PantoA.Z) ;
%QB156:= 	EsitoAccodamento;



(*-----------RESTITUZIONE DEI CANALI Linearizzati ------*)
%QD158:=	FC_SiemensReal2Dword(reale1:= Ist_MapE.GradBraccio) ;(*CH1*)
%QD162:=	FC_SiemensReal2Dword(reale1:= Ist_MapE.Z) ;
%QD166:=	FC_SiemensReal2Dword(reale1:= Ist_MapE.EstBraccio) ;
%QD170:=	FC_SiemensReal2Dword(reale1:= (SEL(PantoParE.Globali.Lub1_enable, Ist_MapE.Z_Braccio2, Ist_MapE.GradPolso))) ;

(*-----------RESTITUZIONE DEI CANALI--------*)
%QW178:=ROL (Ist_MapE.RadBraccio_W,8);	(*CH1*)
%QW180:= ROL (Ist_MapE.Z_W,8);			(*CH2*)
%QW182:= ROL (Ist_MapE.EstBraccio_W,8);	(*CH3*)
%QW184:= SEL(PantoParE.Globali.Lub1_enable,  ROL (Ist_MapE.Z2_W,8), ROL (Ist_MapE.RadPolso_W,8)); 	(*CH4*)
%QX186.0:=PantoA.AbilitaRiavvitatura;
%QX186.1:=PantoA.ViteNonSvitabile;
%QB187 := PantoA.Chiave;


(*mapping in caso di TxScrewing*);
IF HeaderE.Cmd.TxScrewingData
THEN
	(*intestazione Mappata nella zona della flangia in corso*)
	ScrewingE.ProgSvitatura:=		%IB157;
	ScrewingE.Id_ViteInviata:=		%IB158;
	ScrewingE.Viti_Totali_Flangia:=	%IB159;
	ScrewingE.FlangiaInviata:= 		%IB160;
	ScrewingE.ProgRiavvitatura:=	%IB161;

	(*Mappati nella zona dati avvitatura*)
	ScrewingE.ID_Chiave:=			%IB162;
	ScrewingE.ProgAvvitatura:=		%IB163;
	ScrewingE.X:=				FC_SiemensREAL(DWORD1:=%ID164);
	ScrewingE.Y:=				FC_SiemensREAL(DWORD1:=%ID168);
	ScrewingE.Z:=				FC_SiemensREAL(DWORD1:=%ID172);
	ScrewingE.TollR:=				FC_SiemensREAL(DWORD1:=%ID176);
	ScrewingE.TollZ:=				FC_SiemensREAL(DWORD1:=%ID180);
	ScrewingE.ZMin:=				FC_SiemensREAL(DWORD1:=%ID184);
	ScrewingE.ZMax:=				FC_SiemensREAL(DWORD1:=%ID188);

	IF ScrewingE.ProgRiavvitatura = 0 THEN
		ScrewingE.ProgRiavvitatura := ScrewingE.ProgAvvitatura;
	END_IF;

	IF %IB156 = 0 THEN (* se la svitatura è disabilitata, imposto a zero il programma svitatura *)
		ScrewingE.ProgSvitatura := 0;
	END_IF;

END_IF
END_FUNCTION_BLOCK
